// TwinCAT 3 PLC project aft_plc_harv_control
// ProgramVersion: 3.1.4026.12
// CompilerDefines: VISU_USEPROPERTYINFO
// libraries:
//   CmpBitmapPool, * (System)
//   Tc2_Standard, * (Beckhoff Automation GmbH)
//   Tc2_System, * (Beckhoff Automation GmbH)
//   Tc2_Utilities, * (Beckhoff Automation GmbH)
//   Tc3_Module, * (Beckhoff Automation GmbH)
//   VisuDialogs, * (System)
//   TcUnit,newest,www.tcunit.org
//   VisuSymbols,newest,System
// project tree:
//   DUTs/Device Level Structures/PD4/ PD4ControlWord.TcDUT, PD4OperationMode.TcDUT, PD4Polarity.TcDUT, PD4StatusWord.TcDUT, ST_PD4_HW.TcDUT, ST_PD4_IN.TcDUT, ST_PD4_OUT.TcDUT
//   DUTs/Device Level Structures/PD6/ PD6ControlWord.TcDUT, PD6OperationMode.TcDUT, PD6Polarity.TcDUT, PD6StatusWord.TcDUT, ST_PD6_IN.TcDUT, ST_PD6_HW.TcDUT, ST_PD6_OUT.TcDUT
//   DUTs/Device Level Structures/SevCon/ SevconControlWord.TcDUT, SevconStatusWord.TcDUT, ST_SEVCON_HW.TcDUT, ST_SEVCON_IN.TcDUT, ST_SEVCON_OUT.TcDUT
//   DUTs/ FrameSelect.TcDUT
//   DUTs/Message Structures/ ST_BINFILLER_MSG.TcDUT, ST_DRIVE_MSG.TcDUT, ST_ERROR_MSG.TcDUT
//   / GlobalTextList.TcGTLO, PlcTask.TcTTO, Visualization Manager.TcVMO (not stored), VISU_TASK.TcTTO
//   GVLs/ CONFIG.TcGVL, HARV.TcGVL, INDEX.TcGVL, IO.TcGVL, MOTORS.TcGVL, UI.TcGVL
//   POUs/Device Level Function Blocks/ FB_HYDRAULIC_VALVE.TcPOU, FB_PD4.TcPOU, FB_PD6.TcPOU, FB_SDO_READ.TcPOU, FB_SEVCON.TcPOU, FB_SDO_WRITE.TcPOU
//   POUs/ FB_READ_HW.TcPOU, FB_WRITE_HW.TcPOU, MAIN.TcPOU
//   POUs/Log Level Function Blocks/ FB_DRIVE_MSG_LOG.TcPOU, FB_ERROR_MSG_LOG.TcPOU, FB_TIMETRACKER.TcPOU
//   POUs/SubSystem Level Function Blocks/ FB_BINFILLER.TcPOU, FB_BIN_MANAGER.TcPOU, FB_CONVEYANCE.TcPOU, FB_DRIVE.TcPOU, FB_TILT.TcPOU
//   POUs/UI Level Function Blocks/ FB_FRAMESELECTOR.TcPOU
//   Test/ FB_DRIVE_TEST.TcPOU, FB_TILT_TEST.TcPOU, PRG_TEST.TcPOU
//   VISUs/ DriveSysTest.TcVIS, Icons.TcIPO (not stored), TiltControlTest.TcVIS
//   VISUs/Harv UI Components/Home Screen Components/ ChassisControls.TcVIS, DriveControls.TcVIS, LeftRobotStatus.TcVIS, RightRobotStatus.TcVIS, RobotStatusPopup.TcVIS
//   VISUs/Harv UI Components/Stats Screen Components/ LeftRobotStats.TcVIS, HarvStats.TcVIS, RightRobotStats.TcVIS
//   VISUs/Harv UI Components/Supervisor Screen Components/ BinFiller.TcVIS, ColorThreshold.TcVIS, Conveyance.TcVIS, LeftRobotControls.TcVIS, RightRobotControls.TcVIS
//   VISUs/Harv UI Components/ Home_Screen.TcVIS, Stats_Screen.TcVIS, StatusBar.TcVIS, Supervisor_Screen.TcVIS
// real-time tasks:
//   TASK PlcTask: cycle T#2ms, priority 20, ADS port 350
//   TASK VISU_TASK: cycle T#200000us, priority 30, ADS port 351
// I/O:
//   DEVICE Device 1 (EtherCAT), AmsNetId 5.123.135.181.2.1
//     Term 5 (EK1200) [EK1200-5000 EtherCAT Power supply (2A E-Bus)]
//       Term 9 (EL3064) [EL3064 4Ch. Ana. Input 0-10V] (disabled)
//       Term 6 (EL1018) [EL1018 8Ch. Dig. Input 24V, 10µs]
//       Term 7 (EL2008) [EL2008 8Ch. Dig. Output 24V, 0.5A]
//       Term 12 (EL6751) [EL6751 CANopen Master] (disabled)
//       Term 11 (EK1110) [EK1110 EtherCAT extension]
//     Left Steering (PD4-E601L42-E-65-1) [PD4-Ex-E-65-1 EtherCAT Drive (CoE)] (disabled)
//     Right Steering (PD4-E601L42-E-65-1) [PD4-Ex-E-65-1 EtherCAT Drive (CoE)] (disabled)
//   DEVICE Device 2 (EL6751) (disabled), AmsNetId 5.123.135.181.3.1
//     Drive Right (BorgWarner Gen4 (PMAC)Thu Feb  3 22:00:)
//     Drive Left (BorgWarner Gen4 (PMAC)Thu Feb  3 22:00:)
// variable links:
//   aft_plc_harv_control/aft_plc_harv_control Instance <-> Device 1 (EtherCAT)/Left Steering (PD4-E601L42-E-65-1)
//     PlcTask Inputs/MOTORS.SteerLeft.ActualPosition <-> Transmit PDO 1 Mapping Parameter/Position actual value
//     PlcTask Inputs/MOTORS.SteerLeft.OperationModeDisplay <-> Transmit PDO 1 Mapping Parameter/Modes of operation display
//     PlcTask Inputs/MOTORS.SteerLeft.StatusWord <-> Transmit PDO 1 Mapping Parameter/Statusword
//     PlcTask Outputs/MOTORS.SteerLeft.Accel <-> Receive PDO 2 Mapping Parameter/Accel
//     PlcTask Outputs/MOTORS.SteerLeft.ControlWord <-> Receive PDO 1 Mapping Parameter/Controlword
//     PlcTask Outputs/MOTORS.SteerLeft.Decel <-> Receive PDO 2 Mapping Parameter/Decel
//     PlcTask Outputs/MOTORS.SteerLeft.HomingMethod <-> Receive PDO 1 Mapping Parameter/Homing Method
//     PlcTask Outputs/MOTORS.SteerLeft.OperationMode <-> Receive PDO 1 Mapping Parameter/Modes of operation
//     PlcTask Outputs/MOTORS.SteerLeft.Polarity <-> Receive PDO 1 Mapping Parameter/Polarity
//     PlcTask Outputs/MOTORS.SteerLeft.ProfileVelocity <-> Receive PDO 2 Mapping Parameter/Profile velocity
//     PlcTask Outputs/MOTORS.SteerLeft.SubmodeSelect <-> Receive PDO 1 Mapping Parameter/Motor drive submode select
//     PlcTask Outputs/MOTORS.SteerLeft.TargetPosition <-> Receive PDO 2 Mapping Parameter/Target Position
//     PlcTask Outputs/MOTORS.SteerLeft.TargetVelocity <-> Receive PDO 3 Mapping Parameter/vl target velocity
//   aft_plc_harv_control/aft_plc_harv_control Instance <-> Device 1 (EtherCAT)/Right Steering (PD4-E601L42-E-65-1)
//     PlcTask Inputs/MOTORS.SteerRight.ActualPosition <-> Transmit PDO 1 Mapping Parameter/Position actual value
//     PlcTask Inputs/MOTORS.SteerRight.OperationModeDisplay <-> Transmit PDO 1 Mapping Parameter/Modes of operation display
//     PlcTask Inputs/MOTORS.SteerRight.StatusWord <-> Transmit PDO 1 Mapping Parameter/Statusword
//     PlcTask Outputs/MOTORS.SteerRight.Accel <-> Receive PDO 2 Mapping Parameter/Accel
//     PlcTask Outputs/MOTORS.SteerRight.ControlWord <-> Receive PDO 1 Mapping Parameter/Controlword
//     PlcTask Outputs/MOTORS.SteerRight.Decel <-> Receive PDO 2 Mapping Parameter/Decel
//     PlcTask Outputs/MOTORS.SteerRight.HomingMethod <-> Receive PDO 1 Mapping Parameter/Homing Method
//     PlcTask Outputs/MOTORS.SteerRight.OperationMode <-> Receive PDO 1 Mapping Parameter/Modes of operation
//     PlcTask Outputs/MOTORS.SteerRight.Polarity <-> Receive PDO 1 Mapping Parameter/Polarity
//     PlcTask Outputs/MOTORS.SteerRight.ProfileVelocity <-> Receive PDO 2 Mapping Parameter/Profile velocity
//     PlcTask Outputs/MOTORS.SteerRight.SubmodeSelect <-> Receive PDO 1 Mapping Parameter/Motor drive submode select
//     PlcTask Outputs/MOTORS.SteerRight.TargetPosition <-> Receive PDO 2 Mapping Parameter/Target Position
//     PlcTask Outputs/MOTORS.SteerRight.TargetVelocity <-> Receive PDO 3 Mapping Parameter/vl target velocity
//   aft_plc_harv_control/aft_plc_harv_control Instance <-> Device 1 (EtherCAT)/Term 5 (EK1200)/Term 6 (EL1018)
//     PlcTask Inputs/IO.DI_SLICE_0[{0..7}] <-> Channel {1..8}/Input  (8 links)
//   aft_plc_harv_control/aft_plc_harv_control Instance <-> Device 1 (EtherCAT)/Term 5 (EK1200)/Term 7 (EL2008)
//     PlcTask Outputs/IO.DO_SLICE_0[{0..7}] <-> Channel {1..8}/Output  (8 links)
//   aft_plc_harv_control/aft_plc_harv_control Instance <-> Device 1 (EtherCAT)/Term 5 (EK1200)/Term 9 (EL3064)
//     PlcTask Inputs/IO.AI_SLICE_0[{0..3}] <-> AI Standard Channel {1..4}/Value  (4 links)
//   aft_plc_harv_control/aft_plc_harv_control Instance <-> Device 2 (EL6751)/Drive Left (BorgWarner Gen4 (PMAC)Thu Feb  3 22:00:)
//     PlcTask Inputs/MOTORS.DriveLeft.ActualVelocity <-> TxPDO 1/Inputs/Actual Velocity
//     PlcTask Inputs/MOTORS.DriveLeft.AnalogIn{1..4} <-> TxPDO 3/Inputs/Analog In {1..4}  (4 links)
//     PlcTask Inputs/MOTORS.DriveLeft.BatteryCurrent <-> TxPDO 2/Inputs/Battery Current
//     PlcTask Inputs/MOTORS.DriveLeft.BatteryVoltage <-> TxPDO 2/Inputs/Battery Voltage
//     PlcTask Inputs/MOTORS.DriveLeft.CapacitorVoltage <-> TxPDO 2/Inputs/Capacitor Voltage
//     PlcTask Inputs/MOTORS.DriveLeft.HeatsinkTemp <-> TxPDO 2/Inputs/Heatsink Temp
//     PlcTask Inputs/MOTORS.DriveLeft.StatusWord <-> TxPDO 1/Inputs/Status Word
//     PlcTask Outputs/MOTORS.DriveLeft.BrakeOutput <-> RxPDO 3/Outputs/Brake
//     PlcTask Outputs/MOTORS.DriveLeft.ContactorOutput <-> RxPDO 3/Outputs/Power Contactor
//     PlcTask Outputs/MOTORS.DriveLeft.ControlWord <-> RxPDO 1/Outputs/Control Word
//     PlcTask Outputs/MOTORS.DriveLeft.TargetVelocity <-> RxPDO 1/Outputs/Target Velocity

CONFIGURATION aft_plc_harv_control
    RESOURCE PLC ON TwinCAT3
        TASK PlcTask(INTERVAL := T#2ms, PRIORITY := 20);
        TASK VISU_TASK(INTERVAL := T#200000us, PRIORITY := 30);
        PROGRAM MAIN WITH PlcTask : MAIN;
        PROGRAM PRG_TEST WITH PlcTask : PRG_TEST;
        PROGRAM VisuElems_Visu_Prg WITH VISU_TASK : VisuElems.Visu_Prg;
    END_RESOURCE
END_CONFIGURATION

// ---- DUTs/Device Level Structures/PD4/PD4ControlWord.TcDUT
{attribute 'qualified_only'}
{attribute 'strict'}
TYPE PD4ControlWord :
(
	Shutdown := 6,					// 2#0000_0110	
	SwitchOn := 7,					// 0xxx 0111 (Trasition from Ready to Switch On -> Switched On)
	SwitchOnOperationEnable := 15,	// 0xxx 1111 (Switch On and Enable Operation)
	StartHoming:= 16,
	PulseInhibit := 0,				// 0xxx xx0x (activate quick stop and disable)
	QuickStop := 2,					// 0xxx x01x
	DisableOperation := 7,			// 0xxx 0111 (Transition from OpEnable -> Switched On)
	EnableOperation := 2#00101111,			// 0x1x 1111
	FaultReset := 128,				// 1xxx xxxx
	StartMove := 2#00010000,				// xxx1 1111
	AbsoluteMotion := 2#00100000
	// Positive := 64,					// x1xx xxxx
	// Negative :=	0					// x0xx xxxx
)BYTE;
END_TYPE

// ---- DUTs/Device Level Structures/PD4/PD4OperationMode.TcDUT
{attribute 'qualified_only'}
{attribute 'strict'}
TYPE PD4OperationMode :
(
	ProfilePositionMode := 1,
	VelocityMode := 2,
	ProfileVelocityMode := 3,
	ProfileTorqueMode := 4,
	HomingMode := 6,
	CyclicSyncPositionMode := 8
)SINT;
END_TYPE

// ---- DUTs/Device Level Structures/PD4/PD4Polarity.TcDUT
{attribute 'qualified_only'}
{attribute 'strict'}
TYPE PD4Polarity :
(
	Positive := 64,
	Negative := 0
)USINT;
END_TYPE

// ---- DUTs/Device Level Structures/PD4/PD4StatusWord.TcDUT
{attribute 'qualified_only'}
{attribute 'strict'}
TYPE PD4StatusWord :
(
	NotReadyToSwitchOn := 0,	// x0xx 0000
	SwitchOnDisabled := 64,		// x1xx 0000
	ReadyToSwitchOn := 33,		// 1000 0010 0011 0001 (0x8231)
	SwitchedOn := 35,			// 1000 0010 0011 0011 (0x8233)
	OperationEnabled := 39,		// x01x 0111
	QuickStopActive := 7,		// x00x 0111
	Fault := 8,					// x0xx 1000
	TargetReached := 1024,		// 0000 0100 0000 0000 (bit 10)
	HomingComplete := 5120,		// 0001 0100 0000 0000 (bit 10 and 12)
	TargetPositionAccepted := 4096		
)UINT;
END_TYPE

// ---- DUTs/Device Level Structures/PD4/ST_PD4_HW.TcDUT
TYPE ST_PD4_HW :
STRUCT
	StatusWord 				AT %I* : UINT; 
	OperationModeDisplay 	AT %I* : SINT;
	ActualPosition 			AT %I* : DINT;
	ActualVelocity 			AT %I* : INT;
	
	
	ControlWord 	AT %Q* : UINT;
	HomingMethod 	AT %Q* : USINT;
	TargetVelocity 	AT %Q* : INT;
	ProfileVelocity AT %Q* : UDINT;
	Accel 			AT %Q* : UDINT;				
	Decel 			AT %Q* : UDINT;				
	SubmodeSelect	AT %Q* : UDINT;	
	OperationMode 	AT %Q* : SINT;	
	TargetPosition 	AT %Q* : DINT;		
	Polarity 		AT %Q* : USINT;		
END_STRUCT
END_TYPE

// ---- DUTs/Device Level Structures/PD4/ST_PD4_IN.TcDUT
TYPE ST_PD4_IN :
STRUCT
	StatusWord 				: UINT;
	ActualPosition 			: DINT;
	ActualVelocity 			: REAL;
	OperationModeDisplay 	: SINT;
END_STRUCT
END_TYPE

// ---- DUTs/Device Level Structures/PD4/ST_PD4_OUT.TcDUT
TYPE ST_PD4_OUT :
STRUCT
	ControlWord 	: UINT;
	HomingMethod 	: USINT;
	TargetVelocity 	: INT;		// target velocity while in profile velocity mode
	ProfileVelocity : UDINT;	// target velocity while in profile position mode
	Accel 			: UDINT;
	Decel 			: UDINT;
	TargetPosition	: DINT;
	SubmodeSelect 	: UDINT;
	OperationMode 	: SINT;
	Polarity		: USINT;
END_STRUCT
END_TYPE

// ---- DUTs/Device Level Structures/PD6/PD6ControlWord.TcDUT
{attribute 'qualified_only'}
{attribute 'strict'}
TYPE PD6ControlWord :
(
	Shutdown := 6,					// 2#0000_0110	
	SwitchOn := 7,					// 0xxx 0111 (Trasition from Ready to Switch On -> Switched On)
	SwitchOnOperationEnable := 15,	// 0xxx 1111 (Switch On and Enable Operation)
	StartHoming:= 16,
	PulseInhibit := 0,				// 0xxx xx0x (activate quick stop and disable)
	QuickStop := 2,					// 0xxx x01x
	DisableOperation := 7,			// 0xxx 0111 (Transition from OpEnable -> Switched On)
	EnableOperation := 15,			// 0xxx 1111
	FaultReset := 128,				// 1xxx xxxx
	StartMove := 2#00010000,				// xxx1 1111
	AbsoluteMotion := 2#00100000			// xxx1 1111
	// Positive := 64,					// x1xx xxxx
	// Negative :=	0					// x0xx xxxx
)BYTE;
END_TYPE

// ---- DUTs/Device Level Structures/PD6/PD6OperationMode.TcDUT
{attribute 'qualified_only'}
{attribute 'strict'}
TYPE PD6OperationMode :
(
	ProfilePositionMode := 1,
	VelocityMode := 2,
	ProfileVelocityMode := 3,
	ProfileTorqueMode := 4,
	HomingMode := 6,
	CyclicSyncPositionMode := 8
)SINT;
END_TYPE

// ---- DUTs/Device Level Structures/PD6/PD6Polarity.TcDUT
{attribute 'qualified_only'}
{attribute 'strict'}
TYPE PD6Polarity :
(
	Positive := 64,
	Negative := 0
)USINT;
END_TYPE

// ---- DUTs/Device Level Structures/PD6/PD6StatusWord.TcDUT
{attribute 'qualified_only'}
{attribute 'strict'}
TYPE PD6StatusWord :
(
	NotReadyToSwitchOn := 0,	// x0xx 0000
	SwitchOnDisabled := 64,		// x1xx 0000
	ReadyToSwitchOn := 33,		// 1000 0010 0011 0001 (0x8231)
	SwitchedOn := 35,			// 1000 0010 0011 0011 (0x8233)
	OperationEnabled := 39,		// x01x 0111
	QuickStopActive := 7,		// x00x 0111
	Fault := 8,					// x0xx 1000
	TargetReached := 1024,		// 0000 0100 0000 0000 (bit 10)
	HomingComplete := 5120,		// 0001 0100 0000 0000 (bit 10 and 12)
	TargetPositionAccepted := 4096		
)UINT;
END_TYPE

// ---- DUTs/Device Level Structures/PD6/ST_PD6_IN.TcDUT
TYPE ST_PD6_IN :
STRUCT
	StatusWord 				: UINT; 
	OperationModeDisplay 	: SINT;
	ActualPosition 			: DINT;
	ActualVelocity 			: INT;
	ActiveCurrent			: REAL;
END_STRUCT
END_TYPE

// ---- DUTs/Device Level Structures/PD6/ST_PD6_HW.TcDUT
TYPE ST_PD6_HW :
STRUCT
	StatusWord 				AT %I* : UINT; 
	OperationModeDisplay 	AT %I* : SINT;
	ActualPosition 			AT %I* : DINT;
	ActualVelocity 			AT %I* : INT;
	
	
	ControlWord 	AT %Q* : UINT;
	HomingMethod 	AT %Q* : USINT;
	TargetVelocity 	AT %Q* : INT;
	ProfileVelocity AT %Q* : UDINT;
	Accel 			AT %Q* : UDINT;				
	Decel 			AT %Q* : UDINT;				
	SubmodeSelect	AT %Q* : UDINT;	
	OperationMode 	AT %Q* : SINT;	
	TargetPosition 	AT %Q* : DINT;		
	Polarity 		AT %Q* : USINT;		
END_STRUCT
END_TYPE

// ---- DUTs/Device Level Structures/PD6/ST_PD6_OUT.TcDUT
TYPE ST_PD6_OUT :
STRUCT
	ControlWord 	: UINT;
	HomingMethod 	: USINT;
	TargetVelocity 	: INT;
	ProfileVelocity : UDINT;
	Accel 			: UDINT;				
	Decel 			: UDINT;				
	SubmodeSelect	: UDINT;	
	OperationMode 	: SINT;	
	TargetPosition 	: DINT;		
	Polarity 		: USINT;	
END_STRUCT
END_TYPE

// ---- DUTs/Device Level Structures/SevCon/SevconControlWord.TcDUT
{attribute 'qualified_only'}
{attribute 'strict'}
TYPE SevconControlWord :
(
	Shutdown			:= 2#00000110,
	SwitchOn			:= 2#00000111,
	DisableVoltage		:= 2#00000000,
	QuickStop			:= 2#00000010,
	DisableOperation	:= 2#00000111,
	EnableOperation		:= 2#00001111,
	FaultReset			:= 2#00010000
)BYTE;
END_TYPE

// ---- DUTs/Device Level Structures/SevCon/SevconStatusWord.TcDUT
{attribute 'qualified_only'}
{attribute 'strict'}
TYPE SevconStatusWord :
(
	SwitchOnDisabled	:= 2#01000000,
	ReadyToSwitchon		:= 2#00100001,
	Switchedon			:= 2#00100011,
	OperationEnabled	:= 2#00100111,
	QuickStopActive		:= 2#00000111,
	FaultReactionActive	:= 2#00001111,
	Fault				:= 2#00001000
)BYTE;
END_TYPE

// ---- DUTs/Device Level Structures/SevCon/ST_SEVCON_HW.TcDUT
TYPE ST_SEVCON_HW :
STRUCT
	(*Inputs to PLC from Sevcon*)
	StatusWord 				AT %I* : UINT;
	OperationModeDisplay 	AT %I* : SINT;
	ActualVelocity 			AT %I* : UDINT;
	BatteryVoltage			AT %I* : UINT;
	BatteryCurrent			AT %I* : UINT;
	CapacitorVoltage		AT %I* : UINT;
	HeatsinkTemp			AT %I* : USINT;
	AnalogIn1				AT %I* : UINT;
	AnalogIn2				AT %I* : UINT;
	AnalogIn3				AT %I* : UINT;
	AnalogIn4				AT %I* : UINT;
	
	
	(*Outputs to Sevcon from PLC*)
	ControlWord 	AT %Q* : UINT;
	OperationMode 	AT %Q* : SINT;
	TargetVelocity	AT %Q* : UDINT;
	Accel			AT %Q* : UINT;
	Decel			AT %Q* : UINT;
	BrakeOutput		AT %Q* : UINT;
	ContactorOutput	AT %Q* : UINT;
END_STRUCT
END_TYPE

// ---- DUTs/Device Level Structures/SevCon/ST_SEVCON_IN.TcDUT
TYPE ST_SEVCON_IN :
STRUCT
	StatusWord 				: UINT;
	OperationModeDisplay 	: SINT;
	ActualVelocity 			: UDINT;
	BatteryVoltage			: UINT;
	BatteryCurrent			: UINT;
	CapacitorVoltage		: UINT;
	HeatsinkTemp			: UINT;
	AnalogIn1				: UINT;
	AnalogIn2				: UINT;
	AnalogIn3				: UINT;
	AnalogIn4				: UINT;
END_STRUCT
END_TYPE

// ---- DUTs/Device Level Structures/SevCon/ST_SEVCON_OUT.TcDUT
TYPE ST_SEVCON_OUT :
STRUCT
	ControlWord 	: UINT;
	OperationMode 	: SINT;
	TargetVelocity	: UDINT;
	Accel			: UINT;
	Decel			: UINT;
	BrakeOutput		: UINT;
	ContactorOutput	: UINT;
	PreCharge		: UINT;
END_STRUCT
END_TYPE

// ---- DUTs/FrameSelect.TcDUT
{attribute 'qualified_only'}
{attribute 'strict'}
TYPE FrameSelect :
(
	Status	:= 1,
	Warning := 2,
	Error	:= 3
)INT;
END_TYPE

// ---- DUTs/Message Structures/ST_BINFILLER_MSG.TcDUT
{attribute 'pack_mode' := '1'}
TYPE ST_BINFILLER_MSG :
STRUCT
END_STRUCT
END_TYPE

// ---- DUTs/Message Structures/ST_DRIVE_MSG.TcDUT
{attribute 'pack_mode' := '1'}
TYPE ST_DRIVE_MSG :
STRUCT
	TimeStamp			: DT;
	LeftVelocity		: INT;
	RightVelocity		: INT;
	LeftSteeringAngle	: LREAL;
	RightSteeringAngle	: LREAL;
	LeftCurrent			: REAL;
	RightCurrent		: REAL;
	LeftStatusCode		: UINT;
	RightStatusCode		: UINT;
END_STRUCT
END_TYPE

// ---- DUTs/Message Structures/ST_ERROR_MSG.TcDUT
{attribute 'pack_mode' := '1'}
TYPE ST_ERROR_MSG :
STRUCT
	Timestamp	: DT;
	Location	: STRING;
	ErrorCode	: INT;
	Description	: STRING;
END_STRUCT
END_TYPE

// ---- GVLs/CONFIG.TcGVL
{attribute 'qualified_only'}
VAR_GLOBAL
	
	DriveWheelWidth			: REAL := 8.0;
	
	SteeringWheelWidth		: REAL := 5.0;
	WheelBase				: REAL := 137.0;		// Distance between the drive wheels and steering wheels center to center
	FrontTrackWidth			: REAL := 60;		// Distance between the two drive wheels center to center
	RearTrackWidth			: REAL := 72;		// inches
	CasterOffset			: REAL := 8.0;		// Distance between wheel center and rotation center on the steering axes
	
	SevCon_Port				: ARRAY[0..1] OF WORD := [16#1001, 16#1002];	// Drive Right, Drive Left
END_VAR

// ---- GVLs/HARV.TcGVL
{attribute 'qualified_only'}
VAR_GLOBAL
	(*Log Level Function Blocks*)
	ErrorLog	: FB_ERROR_MSG_LOG;
	DriveLog	: FB_DRIVE_MSG_LOG;
	TimeTracker	: FB_TIMETRACKER;
	
	(*SubSystem Level Function Blocks*)
	DriveSys	: FB_DRIVE;
	TiltControl	: FB_TILT;
	BinFiller	: FB_BINFILLER;
	BinManager	: FB_BIN_MANAGER;
	Conveyance	: FB_CONVEYANCE;
	
	(*Device Level Function Blocks*)
	ReadHw		: FB_READ_HW;
	WriteHw		: FB_WRITE_HW;
	
	(*System Level Function Blocks*)
	SystemReboot	: NT_REBOOT;
END_VAR

// ---- GVLs/INDEX.TcGVL
{attribute 'qualified_only'}
VAR_GLOBAL
	(*SEVCON Indexes that will likely be used by the SDO Read/Write function blocks*)
	SpeedControlGains	: DWORD := 16#4651;
	PasswordEntry		: DWORD := 16#5000;
	PasswordKey			: DWORD := 16#5001;	
	NmtState			: DWORD := 16#5110;
	PreChargeActivate	: DWORD := 16#5180;
	FinalPreChargeLevel	: DWORD := 16#5820;
	MinPreChargeLevel	: DWORD := 16#5821;
END_VAR

// ---- GVLs/IO.TcGVL
{attribute 'qualified_only'}
VAR_GLOBAL
	AI_SLICE_0 AT %I* : ARRAY[0..3] OF INT;
	DI_SLICE_0 AT %I* : ARRAY[0..7] OF BOOL;
	
	DO_SLICE_0 AT %Q* : ARRAY[0..7] OF BOOL;
END_VAR

// ---- GVLs/MOTORS.TcGVL
{attribute 'qualified_only'}
VAR_GLOBAL
	DriveLeft	: ST_SEVCON_HW;
	DriveRight	: ST_SEVCON_HW;
//	DriveLeft	: ST_PD6_HW;
//	DriveRight	: ST_PD6_HW;
//	SteerLeft_PD6	: ST_PD6_HW;
//	SteerRight_PD6	: ST_PD6_HW;
	SteerLeft	: ST_PD4_HW;
	SteerRight	: ST_PD4_HW;
END_VAR

// ---- GVLs/UI.TcGVL
{attribute 'qualified_only'}
VAR_GLOBAL
	FrameSelector	: FB_FRAMESELECTOR;
	PickButton		: BOOL;
	EStop			: BOOL;
END_VAR

// ---- POUs/MAIN.TcPOU
PROGRAM MAIN
VAR
	Error			: BOOL;
	SystemReboot	: NT_REBOOT;
	Reboot			: BOOL;
	MsgUpdateTimer	: TON;
	MsgUpdatePeriod	: TIME := T#50MS;
	TimerResetDelay	: INT := 25;
	TimerResetCounter	: INT;
	Version			: REAL := 1.0;
	
	State			: (DEFAULT, INIT, IDLE, RUN, ERROR);
	PrevState		: (DEFAULT, INIT, IDLE, RUN, ERROR);
	StateEntry 		: BOOL;
END_VAR

Harv.ReadHw();

MsgUpdateTimer.PT := MsgUpdatePeriod;

IF PrevState <> State THEN
	StateEntry := TRUE;
	PrevState := State;
ELSE
	StateEntry := FALSE;
END_IF

CASE State OF
	DEFAULT:
		//
	INIT:
		//
	IDLE:
		//
	RUN:
		//
	ERROR:
		//
END_CASE

//IF Error THEN
//	HARV.ErrorLog.AddMsg(TimeStamp := Harv.TimeTracker.TimeStamp, Location := 'MAIN', ErrorCode := 1234, Description := 'TEST');
//	Error := FALSE;
//END_IF

IF MsgUpdateTimer.Q THEN
	TimerResetCounter := TimerResetCounter + 1;
	IF TimerResetCounter = TimerResetDelay THEN
		TimerResetCounter := 0;
		MsgUpdateTimer.IN := FALSE;
	END_IF
ELSE
	TimerResetCounter := 0;
	MsgUpdateTimer.IN := TRUE;
END_IF

SystemReboot(NETID := '', START := Reboot);

MsgUpdateTimer();
Harv.TimeTracker();
Harv.DriveSys();
Harv.TiltControl();
Harv.WriteHw();

END_PROGRAM

// ---- Test/PRG_TEST.TcPOU
PROGRAM PRG_TEST
VAR
	Drive_Test	: FB_DRIVE_TEST;
END_VAR

TcUnit.RUN();

END_PROGRAM

// ---- Test/FB_DRIVE_TEST.TcPOU
FUNCTION_BLOCK FB_DRIVE_TEST EXTENDS TcUnit.FB_TestSuite
VAR_INPUT
END_VAR
VAR_OUTPUT
END_VAR
VAR
END_VAR

SteerAngleTest();
DiffDriveTest();

METHOD DiffDriveTest : REFERENCE TO FB_Test
VAR
	
END_VAR
TEST('DifferentialDriveTest');



TEST_FINISHED();
END_METHOD

METHOD SteerAngleTest : REFERENCE TO FB_Test
VAR
	Drive	: FB_DRIVE;
	AngleInput			: LREAL := 45;
	LeftAngleCalc		: LREAL;
	RightAngleCalc		: LREAL;	
	LeftAngleExpected	: LREAL := 38.89;
	RightAngleExpected	: LREAL := 51.03;
END_VAR
TEST('SteerAngleTest');

(*Zero Steering Angle*)
Drive.CalcWheelAngle(0);
LeftAngleCalc := Drive.SteerLeftAngleTest;
RightAngleCalc := Drive.SteerRightAngleTest;
			
AssertEquals_LREAL(Expected := 0,
				Actual := LeftAngleCalc,
				Delta := 0.1,
				Message := 'Left Angle 0 Calculation Incorrect');
				
AssertEquals_LREAL(Expected := 0,
				Actual := RightAngleCalc,
				Delta := 0.1,
				Message := 'Right Angle 0 Calculation Incorrect');

(*45 Degree Steering Angle*)				
Drive.CalcWheelAngle(AngleInput);
LeftAngleCalc := Drive.SteerLeftAngleTest;
RightAngleCalc := Drive.SteerRightAngleTest;

AssertEquals_LREAL(Expected := LeftAngleExpected,
				Actual := LeftAngleCalc,
				Delta := 0.1,
				Message := 'Left Angle 45 Calculation Incorrect');
				
AssertEquals_LREAL(Expected := RightAngleExpected,
				Actual := RightAngleCalc,
				Delta := 0.1,
				Message := 'Right Angle 45 Calculation Incorrect');

(*-45 Degree Steering Angle*)			
Drive.CalcWheelAngle(-AngleInput);
LeftAngleCalc := Drive.SteerLeftAngleTest;
RightAngleCalc := Drive.SteerRightAngleTest;

AssertEquals_LREAL(Expected := -RightAngleExpected,
				Actual := LeftAngleCalc,
				Delta := 0.1,
				Message := 'Left Angle -45 Calculation Incorrect');
				
AssertEquals_LREAL(Expected := -LeftAngleExpected,
				Actual := RightAngleCalc,
				Delta := 0.1,
				Message := 'Right Angle -45 Calculation Incorrect');
				
(*Positive Max Steering Angle*)

(*Negative Max Steering Angle*)

(*Positive Out of Range Steering Angle*)

(*Negative Out of Range Steering Angle*)
			
TEST_FINISHED();
END_METHOD

END_FUNCTION_BLOCK

// ---- POUs/SubSystem Level Function Blocks/FB_DRIVE.TcPOU
FUNCTION_BLOCK FB_DRIVE
VAR_INPUT
	DriveLeftIN			: ST_SEVCON_IN;
	DriveRightIN		: ST_SEVCON_IN;
//	SteerLeftIN			: ST_PD6_IN;
//	SteerRightIN		: ST_PD6_IN;
	SteerLeftIN			: ST_PD4_IN;
	SteerRightIN		: ST_PD4_IN;
	
	JoyStick_X			: INT;
	JoyStick_Y			: INT;
	JoyStick_Button		: INT;
	ManualDriveEnable	: BOOL;			// Dead man switch on joystick controls
	AutoDriveEnable		: BOOL;			// Likely controlled by python
	ErrorReset			: BOOL;
	
	AutoDriveSpeedCommand	: DINT := 50;
	JohnButtonInput		: BOOL;
END_VAR
VAR_OUTPUT
	DriveLeft	: FB_SEVCON;
	DriveRight	: FB_SEVCON;
//	SteerLeft	: FB_PD6;
//	SteerRight	: FB_PD6;
	SteerLeft	: FB_PD4;
	SteerRight	: FB_PD4;
	
	(*Outputs for unit testing*)
	SteerLeftAngleTest	: LREAL;
	SteerRightAngleTest	: LREAL;

	Error		: BOOL;
	ErrorCode	: INT;
	Ready		: BOOL;
END_VAR
VAR
	State		: (DEFAULT, INIT, IDLE, MANUAL, AUTO, ERROR);
	PrevState	: (DEFAULT, INIT, IDLE, MANUAL, AUTO, ERROR);
	StateEntry 	: BOOL;
	TimeInState	: TIME;
	
	LeftVelCommand	: LREAL;
	LeftVelActual	: LREAL;
	LeftPosActual	: DINT;
	RightVelCommand	: LREAL;
	RightVelActual	: LREAL;
	RightPosActual	: DINT;
	DriveVelInput	: LREAL;
				// Check variable type here, will be in acres / hour
	AutoDriveSpeedActual	: DINT := 45;			// in Acres/hour
	
	SteeringAngleInput		: LREAL;		// unit should be degrees, max range is +/- 89 degrees
	ICC_R					: LREAL;		// instantaneous radius of curvature calculated from steering angle
	LeftWheelAngleCommand	: LREAL;
	LeftWheelAngleActual	: LREAL;
	RightWheelAngleCommand	: LREAL;
	RightWheelAngleActual	: LREAL;
	
	DriveMsgUpdateTimer		: TON;
	DriveMsgUpdatePeriod	: TIME := T#5S;
END_VAR
VAR CONSTANT
	MaxDriveSpeed			: REAL := 1000;		// mm/s
	MaxSteeringAngle		: REAL := 75.0;		// degrees
	JoyStickMaxVal			: INT := 16300;	// raw analog value at extreme
	JoyStickCenter			: INT := 8150;
	DeadBand_X				: INT := 150;		// ~10% or +/- 1V
	DeadBand_Y				: INT := 150;		// ~10% or +/- 1V
	DriveWheelDiameter		: REAL := 762;		// in mm = 30 inches
	DriveWheelEncoderRes	: DINT := 1000;		// was 4000
	DriveWheelGearRatio		: INT := 1;
	SteeringWheelDiameter	: REAL := 660.4;	// in mm = 26 inches
	SteeringEncoderRes		: DINT := 4000;
	SteeringGearRatio		: INT := 14;
	SteeringVel				: UDINT := 500;
	SteeringAcc				: UDINT := 1000;
	SteeringDec				: UDINT := 1000;
	DriveAcc				: UDINT := 1000;
	DriveDec				: UDINT := 10000;
END_VAR

(*DRIVE SYSTEM CONTROL FUNCTION BLOCK
INPUTS:
	- Joystick values in X and Y direction in Manual Drive Mode
	- Deadman switch input for manual mode activation and safety
	- Drive Velocity and Steering Angle from Python in Auto Drive Mode
	- Device status from Sevcons, PD6s and other motion devices

OUTPUTS:
	- Target Velocity commands to SEVCONs for drive speed control
	- Target Position commands to PD6/4s for steering angle control
	- Device status info and function block state*)

IF State <> PrevState THEN
	StateEntry := TRUE;
	PrevState := State;
ELSE
	StateEntry := FALSE;
END_IF

CASE State OF
	DEFAULT:
		IF StateEntry THEN
			TimeInState := T#0MS;
		END_IF
		
		State := INIT;
		
	INIT:
		IF StateEntry THEN
			DriveMsgUpdateTimer.PT := DriveMsgUpdatePeriod;
			TimeInState := T#0MS;
		END_IF
		
		SteerLeft.SetMotionProfile(SteeringVel, SteeringAcc, SteeringDec);
		SteerRight.SetMotionProfile(SteeringVel, SteeringAcc, SteeringDec);
		
		DriveRight.Self := 1;
		DriveLeft.Self := 2;
		
		IF (DriveLeft.Ready) THEN
			Ready := TRUE;
			State := IDLE;
		END_IF
		
//		IF (SteerLeft.Ready AND SteerRight.Ready AND DriveLeft.Ready AND DriveRight.Ready) THEN
//			Ready := TRUE;
//			State := IDLE;
//		END_IF
		
	IDLE:
		IF StateEntry THEN
			TimeInState := T#0MS;
		END_IF
		
		ReadButton();
		
		IF ManualDriveEnable AND Ready THEN
			State := MANUAL;
		ELSIF AutoDriveEnable AND Ready THEN
			State := AUTO;
		END_IF

	MANUAL:
		IF StateEntry THEN
			TimeInState := T#0MS;
			DriveLeft.Enable := TRUE;
			// DriveRight.Enable := TRUE;
			SteerLeft.Enable := TRUE;
			SteerRight.Enable := TRUE;
		END_IF
		
		(*Reads joystick in X direction, scales for steering angle and implements deadband limits*)
		IF (JoyStick_X > (JoyStickCenter + DeadBand_X)) THEN
			SteeringAngleInput := (INT_TO_REAL(JoyStick_X - (JoyStickCenter + DeadBand_X)) / (JoyStickCenter - DeadBand_X)) * MaxSteeringAngle;
		ELSIF (JoyStick_X < (JoyStickCenter - DeadBand_X)) THEN
			SteeringAngleInput := (INT_TO_REAL(JoyStick_X -(JoyStickCenter - DeadBand_X)) / (JoyStickCenter - DeadBand_X)) * MaxSteeringAngle;
		ELSE
			SteeringAngleInput := 0;
		END_IF
		
		(*Reads joystick in Y direction, scales for drive speed and implements deadband limits*)
		IF (JoyStick_Y > (JoyStickCenter + DeadBand_Y)) THEN
			DriveVelInput := (INT_TO_REAL(JoyStick_Y - (JoyStickCenter + DeadBand_Y)) / (JoyStickCenter - DeadBand_Y)) * MaxDriveSpeed;
		ELSIF (JoyStick_Y < (JoyStickCenter - DeadBand_Y)) THEN
			DriveVelInput := (INT_TO_REAL(JoyStick_Y - (JoyStickCenter - DeadBand_Y)) / (JoyStickCenter - DeadBand_Y)) * MaxDriveSpeed;
		ELSE
			DriveVelInput := 0;
		END_IF
		
		(*Calculates wheel angles needed to achieve the commanded steering angle*)
		CalcWheelAngle(SteeringAngleInput);					
		
		(*Calculates differential velocities of the left and right wheels*)
		CalcDiffVelocity(DriveVelInput);				
		
		(*Sets the Sevcon target velocities equal to the calculated values and applies unit scaling*)
		DriveLeft.TargetVelocity := LREAL_TO_UDINT((LeftVelCommand / (3.14 * DriveWheelDiameter)) * DriveWheelGearRatio * DriveWheelEncoderRes);
		DriveRight.TargetVelocity := LREAL_TO_UDINT((RightVelCommand / (3.14 * DriveWheelDiameter)) * DriveWheelGearRatio * DriveWheelEncoderRes);
		
		(*Sets the PD4 steering motors to the correct positions*)
		SteerLeft.TargetPosition := -LREAL_TO_DINT(LeftWheelAngleCommand * ((SteeringEncoderRes * SteeringGearRatio) / 360));		// Negative for motor dir
		SteerRight.TargetPosition := -LREAL_TO_DINT(RightWheelAngleCommand * ((SteeringEncoderRes * SteeringGearRatio) / 360));		// Negative for motor dir
		
		ReadButton();
		
		IF NOT ManualDriveEnable THEN
			DriveLeft.TargetVelocity := 0;
			DriveRight.TargetVelocity := 0;
			DriveLeft.Enable := FALSE;
			DriveRight.Enable := FALSE;
			SteerLeft.Enable := FALSE;
			SteerRight.Enable := FALSE;
			State := IDLE;
		END_IF
		
	AUTO:
		IF StateEntry THEN
			TimeInState := T#0MS;
			DriveLeft.Enable := TRUE;
			DriveRight.Enable := TRUE;
			SteerLeft.Enable := TRUE;
			SteerRight.Enable := TRUE;
		END_IF
		
		(*Calculates wheel angles needed to achieve the commanded steering angle*)
		CalcWheelAngle(SteeringAngleInput);					
		
		(*Calculates differential velocities of the left and right wheels*)
		CalcDiffVelocity(DriveVelInput);	
		
		(*Sets the Sevcon target velocities equal to the calculated values and applies unit scaling*)
		DriveLeft.TargetVelocity := LREAL_TO_UDINT((LeftVelCommand / (3.14 * DriveWheelDiameter)) * DriveWheelGearRatio * DriveWheelEncoderRes);
		DriveRight.TargetVelocity := LREAL_TO_UDINT((RightVelCommand / (3.14 * DriveWheelDiameter)) * DriveWheelGearRatio * DriveWheelEncoderRes);
		
		(*Sets the PD6 steering motors to the correct positions*)
		SteerLeft.TargetPosition := LREAL_TO_DINT(LeftWheelAngleCommand * ((SteeringEncoderRes * SteeringGearRatio) / 360));
		SteerRight.TargetPosition := LREAL_TO_DINT(RightWheelAngleCommand * ((SteeringEncoderRes * SteeringGearRatio) / 360));
		
		IF NOT AutoDriveEnable THEN
			DriveLeft.TargetVelocity := 0;
			DriveRight.TargetVelocity := 0;
			DriveLeft.Enable := FALSE;
			DriveRight.Enable := FALSE;
			SteerLeft.Enable := FALSE;
			SteerRight.Enable := FALSE;
			State := IDLE;
		END_IF
		
	ERROR:
		IF StateEntry THEN
			Error := TRUE;
			Ready := FALSE;
			HARV.ErrorLog.AddMsg(TimeStamp := HARV.TimeTracker.TimeStamp, Location := 'DRIVE', ErrorCode := 9999, Description := 'Drive Test');
			TimeInState := T#0MS;
		END_IF
		
		IF ErrorReset THEN
			DriveLeft.ErrorReset := TRUE;
			DriveRight.ErrorReset := TRUE;
			SteerLeft.ErrorReset := TRUE;
			SteerRight.ErrorReset := TRUE;
			IF (NOT DriveLeft.Error) AND (NOT DriveRight.Error) AND (NOT SteerLeft.Error) AND (NOT SteerRight.Error) THEN
				Error := FALSE;
				ErrorReset := FALSE;
				State := IDLE;
			END_IF
		END_IF
END_CASE

(*Updates Index 0 of the Drive Message Structure with current drive state info*)
//IF DriveMsgUpdateTimer.Q THEN
//	HARV.DriveLog.AddMsg(TimeStamp 			:= HARV.TimeTracker.TimeStamp,
//						LeftVelocity 		:= DriveLeft.PD6_IN.ActualVelocity,
//						LeftSteeringAngle 	:= LeftWheelAngleActual,
//						RightSteeringAngle 	:= RightWheelAngleActual,
//						LeftCurrent 		:= DriveLeft.PD6_IN.ActiveCurrent,
//						LeftStatusCode 		:= DriveLeft.PD6_IN.StatusWord,
//						RightVelocity 		:= DriveRight.PD6_IN.ActualVelocity,
//						RightCurrent 		:= DriveRight.PD6_IN.ActiveCurrent,
//						RightStatusCode 	:= DriveRight.PD6_IN.StatusWord);
//	DriveMsgUpdateTimer.IN := FALSE;
//ELSE
//	DriveMsgUpdateTimer.IN := TRUE;
//END_IF

(*Read actual drive velocities from the SEVCONS in mm/s*)
LeftVelActual := DriveLeft.SEVCON_IN.ActualVelocity;
RightVelActual := DriveRight.SEVCON_IN.ActualVelocity;

(*Read actual wheel positions and calculate actual wheel angles in degrees from steering motors*)
LeftWheelAngleActual := SteerLeft.PD4_IN.ActualPosition;	// Need to convert to degrees
RightWheelAngleActual := SteerRight.PD4_IN.ActualPosition;	// Need to convery to degrees

TimeInState := TimeInState + T#2MS;
//DriveMsgUpdateTimer();
DriveLeft(SEVCON_IN := DriveLeftIN);
DriveRight(SEVCON_IN := DriveRightIN);
SteerLeft(PD4_IN := SteerLeftIN);
SteerRight(PD4_IN := SteerRightIN);

METHOD CalcDiffVelocity : BOOL
VAR_INPUT
	DriveVelInput	: LREAL;
END_VAR
IF SteeringAngleInput <> 0 THEN
	LeftVelCommand := DriveVelInput * (ICC_R + (CONFIG.RearTrackWidth / 2)) / ICC_R;
	RightVelCommand := DriveVelInput * (ICC_R - (CONFIG.RearTrackWidth / 2)) / ICC_R;
ELSE
	LeftVelCommand := DriveVelInput;
	RightVelCommand := DriveVelInput;
END_IF
END_METHOD

METHOD CalcWheelAngle : BOOL
VAR_INPUT
	SteeringAngleInput	: LREAL;		// degrees
END_VAR
VAR
	RightWheelCenterAngle	: LREAL;
	RightSteerCenterAngle	: LREAL;
	LeftWheelCenterAngle	: LREAL;
	LeftSteerCenterAngle	: LREAL;
	EffectiveWheelBase		: REAL;
END_VAR
EffectiveWheelBase := CONFIG.WheelBase + CONFIG.CasterOffset;

IF SteeringAngleInput > MaxSteeringAngle THEN
	ICC_R := CONFIG.WheelBase / TAN(DEG_TO_RAD(MaxSteeringAngle));
ELSIF SteeringAngleInput < -MaxSteeringAngle THEN
	ICC_R := CONFIG.WheelBase / TAN(DEG_TO_RAD(-MaxSteeringAngle));
ELSE
	ICC_R := CONFIG.WheelBase / TAN(DEG_TO_RAD(SteeringAngleInput));		// Calculate radius of curvature relative to the ICC
END_IF

RightWheelCenterAngle := RAD_TO_DEG(ATAN(EffectiveWheelBase/(ICC_R - (CONFIG.FrontTrackWidth / 2)))); 
LeftWheelCenterAngle := RAD_TO_DEG(ATAN(EffectiveWheelBase/(ICC_R + (CONFIG.FrontTrackWidth / 2))));

RightSteerCenterAngle := RAD_TO_DEG(ASIN((CONFIG.CasterOffset)/(SQRT(EXPT((ICC_R - (CONFIG.FrontTrackWidth / 2)),2) + EXPT(EffectiveWheelBase,2)))));
LeftSteerCenterAngle := RAD_TO_DEG(ASIN((CONFIG.CasterOffset)/(SQRT(EXPT((ICC_R + (CONFIG.FrontTrackWidth / 2)),2) + EXPT(EffectiveWheelBase,2)))));

IF SteeringAngleInput < 0 THEN
	RightWheelAngleCommand := RightWheelCenterAngle + RightSteerCenterAngle;
	LeftWheelAngleCommand := LeftWheelCenterAngle + LeftSteerCenterAngle;
ELSE
	RightWheelAngleCommand := RightWheelCenterAngle - RightSteerCenterAngle;
	LeftWheelAngleCommand := LeftWheelCenterAngle - LeftSteerCenterAngle;
END_IF

SteerLeftAngleTest := LeftWheelAngleCommand;
SteerRightAngleTest	:= RightWheelAngleCommand;

//RightWheelAngle := RAD_TO_DEG(ATAN(CONFIG.WheelBase/(ICC_R - (CONFIG.FrontTrackWidth / 2))));
//LeftWheelAngle := RAD_TO_DEG(ATAN(CONFIG.WheelBase/(ICC_R + (CONFIG.FrontTrackWidth / 2))));
END_METHOD

METHOD ReadButton : BOOL
VAR
	SwitchThreshold	: INT := 1000;
	LowThreshold 	: INT := 500;
END_VAR
IF JoyStick_Button > SwitchThreshold THEN
	ManualDriveEnable := FALSE;
ELSIF JoyStick_Button < SwitchThreshold AND JoyStick_Button > LowThreshold THEN
	ManualDriveEnable := TRUE;
ELSE
	//ManualDriveEnable := FALSE;
END_IF
END_METHOD

END_FUNCTION_BLOCK

// ---- POUs/Device Level Function Blocks/FB_SEVCON.TcPOU
FUNCTION_BLOCK FB_SEVCON
VAR_INPUT
	SEVCON_IN 		: ST_SEVCON_IN;
	Enable			: BOOL;
	ErrorReset		: BOOL;
	TargetVelocity	: UDINT;
	Self			: INT;
END_VAR
VAR_OUTPUT
	SEVCON_OUT : ST_SEVCON_OUT;
	Error		: BOOL;
	ErrorCode	: INT;
	Ready		: BOOL;
	Running		: BOOL;
END_VAR
VAR
	State		: (DEFAULT, INIT, SWITCH_ON_DISABLED, READY_TO_SWITCH_ON, SWITCHED_ON, OPERATION_ENABLED, ERROR);
	PrevState 	: (DEFAULT, INIT, SWITCH_ON_DISABLED, READY_TO_SWITCH_ON, SWITCHED_ON, OPERATION_ENABLED, ERROR);
	TimeInState	: TIME;
	StateEntry 	: BOOL;
	SwitchOn	: BOOL;
	SDO_Write		: FB_SDO_WRITE;
	SDO_WriteData	: ARRAY[0..255] OF BYTE;
	SDO_Read		: FB_SDO_READ;
	SDO_ReadData	: ARRAY[0..255] OF BYTE;
	PreChargeTimer	: TON;
	PreChargeDelay	: TIME := T#3S;
	PreChargeActive	: BOOL;
	
	HiSpeedKp		: BYTE;
	HiSpeedKi		: BYTE;
	LoSpeedKp		: BYTE;
	LoSpeedKi		: BYTE;
END_VAR
VAR CONSTANT
	VoltageMult		: REAL := 0.0625;	// Multiply by voltage params for actual voltages
	MinCapVoltage	: REAL := 40.0;		// check w/ Cedric
END_VAR



IF State <> PrevState THEN
	StateEntry := TRUE;
	PrevState := State;
ELSE
	StateEntry := FALSE;
END_IF

CASE State OF
	DEFAULT:
		State := INIT;
		
	INIT:
		// Set initial parameters
		
		Ready := FALSE;
		SEVCON_OUT.ControlWord := SevConControlWord.DisableVoltage;
		PreChargeTimer.PT := PreChargeDelay;
		
		State := SWITCH_ON_DISABLED;
		
		
	SWITCH_ON_DISABLED:
		IF StateEntry THEN
			SEVCON_OUT.ControlWord := SevConControlWord.DisableVoltage;
			SEVCON_OUT.TargetVelocity := 0;
			SEVCON_OUT.ContactorOutput := 0;
			SEVCON_OUT.BrakeOutput := 0;
		END_IF
		
		IF (SEVCON_IN.StatusWord AND SevConStatusWord.SwitchOnDisabled) = SevConStatusWord.SwitchOnDisabled THEN
			SEVCON_OUT.ControlWord := SevConControlWord.Shutdown;
			State := READY_TO_SWITCH_ON;
		END_IF
		
	READY_TO_SWITCH_ON:
		IF StateEntry THEN
			IF (SEVCON_IN.CapacitorVoltage * VoltageMult) < MinCapVoltage THEN
				PreCharge(TRUE);
			END_IF
			PreChargeTimer.IN := TRUE;
		END_IF
		
		IF ((SEVCON_IN.CapacitorVoltage * VoltageMult) > MinCapVoltage) AND PreChargeTimer.Q THEN
			SEVCON_OUT.ContactorOutput := 65535;
			PreCharge(FALSE);
			SwitchOn := TRUE;
			PreChargeTimer.IN := FALSE;
		END_IF
		
		IF SwitchOn AND ((SEVCON_IN.StatusWord AND SevConStatusWord.ReadyToSwitchon) = SevConStatusWord.ReadyToSwitchon) THEN
			SEVCON_OUT.ControlWord := SevConControlWord.SwitchOn;
			State := SWITCHED_ON;
		END_IF
	
	SWITCHED_ON:
		IF StateEntry THEN
			//
		END_IF
		
		IF (SEVCON_IN.StatusWord AND SevConStatusWord.Switchedon) = SevConStatusWord.Switchedon THEN
			Ready := TRUE;
		ELSE
			Ready := FALSE;
		END_IF
		
		IF Enable AND Ready THEN
			SEVCON_OUT.ControlWord := SevConControlWord.EnableOperation;
			State := OPERATION_ENABLED;
		END_IF

	OPERATION_ENABLED:
		IF StateEntry THEN
			SEVCON_OUT.BrakeOutput := 65535;
			Running := TRUE;
		END_IF
		
		IF NOT Enable THEN
			Running := FALSE;
			SEVCON_OUT.TargetVelocity := 0;
			IF SEVCON_IN.ActualVelocity = 0 THEN
				SEVCON_OUT.BrakeOutput := 0;
				SEVCON_OUT.ControlWord := SevConControlWord.DisableOperation;
				State := SWITCHED_ON;
			END_IF
		ELSE
			SEVCON_OUT.TargetVelocity := TargetVelocity;
		END_IF
	
	ERROR:
		IF StateEntry THEN
			Ready := FALSE;
			Error := TRUE;
		END_IF
		
		IF ErrorReset THEN
			SEVCON_OUT.ControlWord := SevConControlWord.FaultReset;
			IF (SEVCON_IN.StatusWord AND SevConStatusWord.Fault) = 0 THEN
				Error := FALSE;
				ErrorReset := FALSE;
				State := SWITCH_ON_DISABLED;
			END_IF
		END_IF
END_CASE

IF (SEVCON_IN.StatusWord AND SevConStatusWord.Fault) = SevConStatusWord.Fault THEN
	State := ERROR;
END_IF

PreChargeTimer();

METHOD PreCharge : BOOL
VAR_INPUT
	Start	: BOOL;
END_VAR
IF Start THEN
	SDO_WriteData[0] := 16#1;
	PreChargeActive := TRUE;
ELSIF NOT Start THEN
	SDO_WriteData[0] := 16#0;
	PreChargeActive := FALSE;
END_IF

SDO_WRITE(ADSNetID := '5.117.40.235.3.1',
		PortNr := CONFIG.SevCon_Port[self-1],
		CO_Index := INDEX.PreChargeActivate,
		CO_SubIndex := 0,
		DataLength := 1,
		StartWriting := TRUE,
		WriteData := SDO_WriteData);
END_METHOD

METHOD WriteTuningValues : BOOL
VAR_INPUT
	KpHi	: BYTE;
	KiHi	: BYTE;
	KpLo	: BYTE;
	KiLo	: BYTE;
END_VAR
END_METHOD

END_FUNCTION_BLOCK

// ---- POUs/Device Level Function Blocks/FB_SDO_WRITE.TcPOU
FUNCTION_BLOCK FB_SDO_WRITE
VAR_INPUT
	ADSNetID		: STRING(23);   			(* The AMSNetID addresses the EL6751. Can be empty if only one local single channel card is present*)
    PortNr			: WORD;           			(* The Port No. addresses the CANopen Node (see System Manager) *)
    CO_Index		: DWORD;        			(* This is the Index of the CANopen Object Dictionary Entry*)
    CO_SubIndex		: DWORD;     				(*This is the Sub-Index of the CANopen Object Dictionary Entry*)
    DataLength		: DWORD;      				(* This is the Length of the CANopen Object Dictionary Entry*)
    StartWriting	: BOOL;     				(*only reset to FALSE after WriteDataFinished=TRUE*)
    WriteData		: ARRAY[0..255] OF BYTE; 	(*This array contains the data to be written to the CANopen Object Dictionary*)
END_VAR
VAR_OUTPUT
	WriteDataFinished	: BOOL;
    Error				: DWORD;
END_VAR
VAR
	state		: BYTE := 0;
    ADSWRITE	: ADSWRITE;
END_VAR

CASE
state OF
    0:
        IF StartWriting THEN
           WriteDataFinished := FALSE;
           Error := 0;
           ADSWrite(
               NETID:= ADSNetID,
               PORT:= PortNr,
               IDXGRP:= CO_Index,
               IDXOFFS:= CO_SubIndex,
               LEN:= DataLength,
               SRCADDR:= ADR(WriteData),
               WRITE:= TRUE,
               TMOUT := T#1s
               );
           IF ADSWrite.err THEN
               state := 2;
               WriteDataFinished := TRUE;
               Error := ADSWrite.ErrId;
           ELSE
               state := 1;
           END_IF
        ELSE
           ADSWrite(
               NETID:= '',
               PORT:= PortNr,
               IDXGRP:= CO_Index,
               IDXOFFS:= CO_SubIndex,
               LEN:= DataLength,
               SRCADDR:= ADR(WriteData),
               WRITE:= FALSE,
               TMOUT := T#1s
               );
        END_IF
    1:
        ADSWrite(WRITE:= FALSE);
        IF ADSWrite.err THEN
           state := 2;
           WriteDataFinished := TRUE;
           Error := ADSWrite.ErrId;
        ELSE
           IF NOT ADSWrite.busy THEN
               state := 2;
               WriteDataFinished := TRUE;
           END_IF
        END_IF
    2:
        ADSWrite(WRITE:= FALSE);
        state := 0;
END_CASE

END_FUNCTION_BLOCK

// ---- POUs/Device Level Function Blocks/FB_SDO_READ.TcPOU
FUNCTION_BLOCK FB_SDO_READ
VAR_INPUT
	ADSNetID:STRING(23); (* The AMSNetID addresses the EL6751. Can be empty if only one local single channel card is present*)
    PortNr:WORD;         (* This Port No. addresses the CANopen Node (see System Manager) *)
    CO_Index:DWORD;      (* This is the Index of the CANopen Object Dictionary Entry*)
    CO_SubIndex:DWORD;   (* This is the Sub-Index of the CANopen Object Dictionary Entry*)
    DataLength:DWORD;    (* This is the Length of the CANopen Object Dictionary Entry*)
    StartReading:BOOL;   (* only reset to FALSE after ReadDataAvailable=TRUE*)
END_VAR
VAR_OUTPUT
	ReadData:ARRAY[0..255] OF BYTE;
    ReadDataAvailable:BOOL;
    Error:DWORD;
END_VAR
VAR
	state:BYTE := 0;
    ADSREAD:ADSREAD;
END_VAR

CASE
state OF
    0:
        IF StartReading THEN
           ReadDataAvailable := FALSE;
           Error := 0;
           ADSRead(
               NETID:= ADSNetID,
               PORT:= PortNr,
               IDXGRP:= CO_Index,
               IDXOFFS:= CO_SubIndex,
               LEN:= DataLength,
               DESTADDR:= ADR(ReadData),
               READ:= TRUE,
               TMOUT := T#1s
               );
           IF ADSRead.err THEN
               state := 2;
               ReadDataAvailable := TRUE;
               Error := ADSRead.ErrId;
           ELSE
               state := 1;
           END_IF
        ELSE
           ADSRead(
               NETID:= ADSNetID,
               PORT:= PortNr,
               IDXGRP:= CO_Index,
               IDXOFFS:= CO_SubIndex,
               LEN:= DataLength,
               DESTADDR:= ADR(ReadData),
               READ:= FALSE,
               TMOUT := T#1s
           );
        END_IF
    1:
        ADSRead(READ:= FALSE);
        IF ADSRead.err THEN
           state := 2;
           ReadDataAvailable := TRUE;
           Error := ADSRead.ErrId;
        ELSE
           IF NOT ADSRead.busy THEN
               state := 2;
               ReadDataAvailable := TRUE;
           END_IF
        END_IF
    2:
        ADSRead(READ:= FALSE);
        state := 0;
END_CASE

END_FUNCTION_BLOCK

// ---- POUs/Device Level Function Blocks/FB_PD4.TcPOU
FUNCTION_BLOCK FB_PD4
VAR_INPUT
	PD4_IN 			: ST_PD4_IN;
	Enable 			: BOOL;
	ErrorReset 		: BOOL;
	TargetVelocity 	: INT;
	TargetPosition	: DINT;			// Check variable type
	Self 			: INT;
END_VAR
VAR_OUTPUT
	PD4_OUT : ST_PD4_OUT;
	Ready 	: BOOL;
	Error	: BOOL;
END_VAR
VAR
//	State 		: DINT;
	State		: (DEFAULT, INIT, SWITCH_ON_DISABLED, READY_TO_SWITCH_ON, SWITCHED_ON, OPERATION_ENABLED, ERROR);
	PrevState 	: (DEFAULT, INIT, SWITCH_ON_DISABLED, READY_TO_SWITCH_ON, SWITCHED_ON, OPERATION_ENABLED, ERROR);
	StateEntry 	: BOOL;
	Homed		: BOOL;
END_VAR

// POWER FSM State Machine for EtherCAT PD4 Control

IF State <> PrevState THEN
	StateEntry := TRUE;
	PrevState := State;
ELSE
	StateEntry := FALSE;
END_IF

CASE State OF
	DEFAULT:
		State := INIT;
		
	INIT:
		Ready := FALSE;
		PD4_OUT.ControlWord := PD4ControlWord.PulseInhibit;
		PD4_OUT.Polarity := PD4Polarity.Positive;
		
		PD4_OUT.OperationMode := PD4OperationMode.HomingMode;
		PD4_OUT.HomingMethod := 35;									// Zero at current position
		PD4_OUT.ControlWord := PD4ControlWord.StartHoming;
		
		IF PD4_IN.ActualPosition = 0 THEN
			SetMode(PD4OperationMode.ProfilePositionMode);
			SetAbsoluteMotion();
//			SetMode(PD4OperationMode.VelocityMode);
			State := SWITCH_ON_DISABLED;
		END_IF

	SWITCH_ON_DISABLED:
		IF StateEntry THEN
			PD4_OUT.ControlWord := PD4ControlWord.PulseInhibit;
			PD4_OUT.TargetVelocity := 0;
		END_IF
		
		IF ((PD4_IN.StatusWord AND PD4StatusWord.SwitchOnDisabled) = PD4StatusWord.SwitchOnDisabled) THEN
			PD4_OUT.ControlWord := PD4ControlWord.Shutdown;
			State := READY_TO_SWITCH_ON;
		END_IF
		
	READY_TO_SWITCH_ON:
		IF ((PD4_IN.StatusWord AND PD4StatusWOrd.ReadyToSwitchOn) = PD4StatusWOrd.ReadyToSwitchOn) THEN
			PD4_OUT.ControlWord := PD4ControlWord.SwitchOn;
			State := SWITCHED_ON;
		END_IF
		
	SWITCHED_ON:
		IF StateEntry THEN
			Ready := TRUE;
		END_IF
		
		IF (((PD4_IN.StatusWord AND PD4StatusWOrd.SwitchedOn) = PD4StatusWOrd.SwitchedOn) AND Enable) THEN
			PD4_OUT.TargetPosition := PD4_IN.ActualPosition;
			PD4_OUT.ControlWord := PD4ControlWord.EnableOperation;
			State := OPERATION_ENABLED;
		END_IF
		
	OPERATION_ENABLED:
		IF StateEntry THEN
			PD4_OUT.TargetPosition := PD4_IN.ActualPosition;
			TargetPosition := PD4_IN.ActualPosition;
		END_IF
		
		PD4_OUT.TargetPosition := TargetPosition;
		ToggleMoveBit();
//		PD4_OUT.TargetVelocity := TargetVelocity;	
		
		IF NOT Enable THEN
//			PD4_OUT.TargetVelocity := 0;
			PD4_OUT.TargetPosition := PD4_IN.ActualPosition;
			PD4_OUT.ControlWord := PD4ControlWord.DisableOperation;
			State := SWITCHED_ON;
		END_IF
		
	ERROR:
		IF StateEntry THEN
			Ready := FALSE;
			Error := TRUE;	
		END_IF
		
		IF ErrorReset THEN
			PD4_OUT.ControlWord := PD4ControlWord.FaultReset;
			IF ((PD4_IN.StatusWord AND PD4StatusWOrd.Fault) = 0) THEN
				Error := FALSE;
				State := SWITCH_ON_DISABLED;
			END_IF
		END_IF
END_CASE

IF ((PD4_IN.StatusWord AND PD4StatusWord.Fault) = PD4StatusWord.Fault) THEN
	State := ERROR;
END_IF

METHOD SetAbsoluteMotion : BOOL
VAR_INPUT
END_VAR
PD4_OUT.ControlWord := PD4_OUT.ControlWord OR PD4ControlWord.AbsoluteMotion;
END_METHOD

METHOD SetMaxCurrent : BOOL
VAR_INPUT
END_VAR
END_METHOD

METHOD SetMode : BOOL
VAR_INPUT
	OperationMode	: PD4OperationMode;
END_VAR
PD4_OUT.OperationMode := OperationMode;
PD4_OUT.SubmodeSelect := 1;
END_METHOD

METHOD SetMotionProfile : BOOL
VAR_INPUT
	Velocity 	: UDINT;
	Accel 		: UDINT;
	Decel 		: UDINT;
END_VAR
PD4_OUT.ProfileVelocity := Velocity;
PD4_OUT.Accel := Accel;
PD4_OUT.Decel := Decel;
END_METHOD

METHOD ToggleMoveBit : BOOL
VAR_INPUT
END_VAR
IF (PD4_OUT.ControlWord AND PD4ControlWord.StartMove) = PD4ControlWord.StartMove THEN
	PD4_OUT.ControlWord := (PD4_OUT.ControlWord AND (NOT PD4ControlWord.StartMove));
ELSE
	PD4_OUT.ControlWord := (PD4_OUT.ControlWord OR PD4ControlWord.StartMove);
END_IF
END_METHOD

END_FUNCTION_BLOCK

// ---- POUs/Log Level Function Blocks/FB_ERROR_MSG_LOG.TcPOU
FUNCTION_BLOCK FB_ERROR_MSG_LOG
VAR
	Buffer 	: ARRAY[0..MaxBufferSize] OF ST_ERROR_MSG;
	Index	: INT;
END_VAR
VAR CONSTANT
	MaxBufferSize	: INT := 1000;
END_VAR

METHOD AddMsg : BOOL
VAR_INPUT
	TimeStamp	: DT;
	Location	: STRING;
	ErrorCode	: INT;
	Description	: STRING;
END_VAR
VAR
	i	: INT;
END_VAR
FOR i := 0 TO MaxBufferSize DO
	IF Buffer[MaxBufferSize - i].Location = '' THEN
		CONTINUE;
	ELSE
		Buffer[MaxBufferSize - i + 1].Location 		:= Buffer[MaxBufferSize - i].Location;
		Buffer[MaxBufferSize - i + 1].TimeStamp 	:= Buffer[MaxBufferSize - i].TimeStamp;
		Buffer[MaxBufferSize - i + 1].ErrorCode 	:= Buffer[MaxBufferSize - i].ErrorCode;
		Buffer[MaxBufferSize - i + 1].Description 	:= Buffer[MaxBufferSize - i].Description;
	END_IF
END_FOR

Buffer[0].Location 		:= Location;
Buffer[0].Timestamp 	:= TimeStamp;
Buffer[0].ErrorCode 	:= ErrorCode;
Buffer[0].Description 	:= Description;

Index := Index + 1;
END_METHOD

END_FUNCTION_BLOCK

// ---- POUs/Log Level Function Blocks/FB_DRIVE_MSG_LOG.TcPOU
FUNCTION_BLOCK FB_DRIVE_MSG_LOG
VAR
	Buffer	: ARRAY[0..MaxBufferSize] OF ST_DRIVE_MSG;
	Index : INT;
END_VAR
VAR CONSTANT
	MaxBufferSize	: INT := 1000;
END_VAR

METHOD AddMsg : BOOL
VAR_INPUT
	TimeStamp			: DT;
	LeftVelocity		: INT;
	RightVelocity		: INT;
	LeftSteeringAngle	: LREAL;
	RightSteeringAngle	: LREAL;
	LeftCurrent			: REAL;
	RightCurrent		: REAL;
	LeftStatusCode		: UINT;
	RightStatusCode		: UINT;
END_VAR
VAR
	i: INT;
END_VAR
FOR i := 0 TO MaxBufferSize DO
	IF Buffer[MaxBufferSize - i].LeftVelocity = 0.0 THEN
		CONTINUE;
	ELSE
		Buffer[MaxBufferSize - i + 1].TimeStamp 			:= Buffer[MaxBufferSize - i].TimeStamp;
		Buffer[MaxBufferSize - i + 1].LeftVelocity 			:= Buffer[MaxBufferSize - i].LeftVelocity;
		Buffer[MaxBufferSize - i + 1].RightVelocity 		:= Buffer[MaxBufferSize - i].RightVelocity;
		Buffer[MaxBufferSize - i + 1].LeftSteeringAngle 	:= Buffer[MaxBufferSize - i].LeftSteeringAngle;
		Buffer[MaxBufferSize - i + 1].RightSteeringAngle 	:= Buffer[MaxBufferSize - i].RightSteeringAngle;
		Buffer[MaxBufferSize - i + 1].LeftCurrent 			:= Buffer[MaxBufferSize - i].LeftCurrent;
		Buffer[MaxBufferSize - i + 1].RightCurrent 			:= Buffer[MaxBufferSize - i].RightCurrent;
		Buffer[MaxBufferSize - i + 1].LeftStatusCode 		:= Buffer[MaxBufferSize - i].LeftStatusCode;
		Buffer[MaxBufferSize - i + 1].RightStatusCode 		:= Buffer[MaxBufferSize - i].RightStatusCode;
	END_IF
END_FOR

Buffer[0].Timestamp 			:= TimeStamp;
Buffer[0].LeftVelocity 			:= LeftVelocity;
Buffer[0].RightVelocity 		:= RightVelocity;
Buffer[0].LeftSteeringAngle 	:= LeftSteeringAngle;
Buffer[0].RightSteeringAngle 	:= RightSteeringAngle;
Buffer[0].LeftCurrent 			:= LeftCurrent;
Buffer[0].RightCurrent 			:= RightCurrent;
Buffer[0].LeftStatusCode 		:= LeftStatusCode;
Buffer[0].RightStatusCode 		:= RightStatusCode;

Index := Index + 1;
END_METHOD

END_FUNCTION_BLOCK

// ---- POUs/Log Level Function Blocks/FB_TIMETRACKER.TcPOU
FUNCTION_BLOCK FB_TIMETRACKER
VAR_INPUT
END_VAR
VAR_OUTPUT
	TimeStamp		: DT;
END_VAR
VAR
	GetSystemTime	: FB_LOCALSYSTEMTIME;
	TimeStampStruct	: TIMESTRUCT;
END_VAR

GetSystemTime(sNetID := '', bEnable := TRUE, systemTime => TimeStampStruct);
TimeStamp := SYSTEMTIME_TO_DT(TimeStampStruct);

END_FUNCTION_BLOCK

// ---- POUs/SubSystem Level Function Blocks/FB_TILT.TcPOU
FUNCTION_BLOCK FB_TILT
VAR_INPUT
	IMU_Roll				: INT;
	IMU_Pitch				: INT;
	AutoTiltControlEnable	: BOOL;
	ManualTiltControlEnable : BOOL;
	StartupEnable			: BOOL;
	TestModeEnable			: BOOL;
	PressureSwitch			: BOOL;
END_VAR
VAR_OUTPUT
	RollValveLeft	: FB_HYDRAULIC_VALVE;
	RollValveRight	: FB_HYDRAULIC_VALVE;
	PitchValve		: FB_HYDRAULIC_VALVE;
	PumpContactor	: BOOL;
	Error			: BOOL;
	ErrorCode		: DINT;
	Ready			: BOOL;
END_VAR
VAR
	TiltDisplacement		: REAL;
	TiltLeftDisplacement	: REAL;
	TiltRightDisplacement	: REAL;
	
	RollAngle				: REAL;
	PitchAngle				: REAL;
	SlopeAngle				: REAL;
	
	State					: (DEFAULT, INIT, IDLE, STARTUP, MANUAL, AUTO, TEST, ERROR);
	PrevState				: (DEFAULT, INIT, IDLE, STARTUP, MANUAL, AUTO, TEST, ERROR);
	StateEntry				: BOOL;
	
	StartHoming				: BOOL;
	Homed					: BOOL;
	CurrentAxis				: INT;
	RearStartPosition		: BOOL;
	FrontStartPosition		: BOOL;
	InStartPosition			: BOOL;
	StartupTimer			: TON;
	StartDelay				: TIME := T#1500MS;
	PumpStartupTimer		: TON;
	PumpStartupDelay		: TIME := T#2000MS;
	CylinderBumpTimer		: TON;
	CylinderBumpDelay		: TIME := T#300MS;
	
	RollAxisLevel			: BOOL;
	PitchAxisLevel			: BOOL;
	
	RollCW_Command			: BOOL;
	RollCCW_Command			: BOOL;
	PitchUp_Command			: BOOL;
	PitchDown_Command		: BOOL;
	Raise_Command			: BOOL;
	Lower_Command			: BOOL;
	Level_Command			: BOOL;
	
	IMU_Roll_Avg			: INT;
	RollDataBuffer			: ARRAY[0..9] OF INT;
	IMU_Pitch_Avg			: INT;
	PitchDataBuffer			: ARRAY[0..9] OF INT;
	
	PressureSwitch_FTRIG	: F_TRIG;
	RearLeftCheck			: BOOL;
	RearRightCheck			: BOOL;
	FrontCheck				: BOOL;
	PitchAngleStart			: REAL;
	RollAngleStart			: REAL;
END_VAR
VAR CONSTANT
	IMU_DeadBand			: INT := 400;
	IMU_Center				: INT := 16535;
	IMU_MaxAngle			: REAL := 30;
	RollControlThreshold	: REAL := 1.0;		// angular delta where the tilt controller kicks in
	PitchControlThreshold	: REAL := 1.0;
	PitchStartupAngle		: REAL := 7.0;		// roughly half stroke on rear cylinders when starting flat
	MaxRollAngle			: REAL := 10;
	MaxPitchAngle			: REAL := 20;
END_VAR



IF State <> PrevState THEN
	StateEntry := TRUE;
	PrevState := State;
ELSE
	StateEntry := FALSE;
END_IF

PressureSwitch_FTRIG.CLK := PressureSwitch;

CASE State OF
	DEFAULT:
		State := INIT;
		
	INIT:
		IF StateEntry THEN
			RearStartPosition := FALSE;
			FrontStartPosition := FALSE;
			InStartPosition := FALSE;
			StartupTimer.PT := StartDelay;
			PumpStartupTimer.PT := PumpStartupDelay;
			CylinderBumpTimer.PT := CylinderBumpDelay;
		END_IF
		
		State := IDLE;
		
	IDLE:
		IF StateEntry THEN
			Hold(TRUE);
		END_IF
		
		IF AutoTiltControlEnable AND InStartPosition THEN
			State := Auto;
		ELSIF ManualTiltControlEnable THEN
			State := MANUAL;
		ELSIF StartupEnable THEN
			State := STARTUP;
		ELSIF TestModeEnable THEN
			State := TEST;
		END_IF
	
	STARTUP:
		IF StateEntry THEN
			PumpContactor := TRUE;
			PumpStartupTimer.IN := TRUE;
			PitchAngleStart := PitchAngle;
			RollAngleStart	:= RollAngle;
		END_IF	
		
		IF PumpStartupTimer.Q THEN
			IF (NOT RearStartPosition) AND (NOT FrontStartPosition) THEN
				RollValveLeft.Extend();
				RollValveRight.Extend();
				IF PitchAngle <= (PitchAngleStart - PitchStartupAngle) THEN
					RollValveLeft.Neutral();
					RolLValveRight.Neutral();
					StartupTimer.IN := FALSE;
					RearStartPosition := TRUE;
				END_IF
			ELSIF( RearStartPosition) AND (NOT FrontStartPosition) THEN
				PitchUp(TRUE);
				IF PitchAngle >= PitchAngleStart THEN
					PitchUp(FALSE);
					FrontStartPosition := TRUE;
					InStartPosition := TRUE;
				END_IF
			END_IF
		END_IF
		
		IF NOT StartupEnable OR InStartPosition THEN
			PumpStartupTimer.IN := FALSE;
			Hold(TRUE);
			PumpContactor := FALSE;
			StartupEnable := FALSE;
			State := IDLE;
		END_IF
	
	MANUAL:	
		IF StateEntry THEN
			PumpContactor := TRUE;
		END_IF
		
		IF RollCW_Command THEN
			RollCW(TRUE);
			IF RollAngle >= 8.0 THEN
				RollCW(FALSE);
				RollCW_Command := FALSE;
			END_IF
		ELSIF RollCCW_Command THEN
			RollCCW(TRUE);
			IF RollAngle <= -8.0 THEN
				RollCCW(FALSE);
				RollCCW_Command := FALSE;
			END_IF
		ELSIF Level_Command THEN
			IF RollAngle > 0 AND NOT RollAxisLevel THEN
				RollCCW(TRUE);
				RollAxisLevel := FALSE;
			ELSIF RollAngle < 0 AND NOT RollAxisLevel THEN
				RollCW(TRUE);
				RollAxisLevel := FALSE;
			ELSE
				RollCW(FALSE);
				RollCCW(FALSE);
				RollAxisLevel := TRUE;
			END_IF
			
			IF PitchAngle > 0 AND RollAxisLevel THEN
				PitchDown(TRUE);
			ELSIF PitchANgle < 0 AND RollAxisLevel THEN
				PitchUp(TRUE);
			ELSE
				PitchValve.Neutral();
				PitchAxisLevel := TRUE;
			END_IF
			
			IF RollAxisLevel AND PitchAxisLevel THEN
				Level_Command := FALSE;
			END_IF
		ELSIF Raise_Command THEN
			Raise(TRUE);
		ELSIF Lower_Command THEN
			Lower(TRUE);
		ELSIF PitchUp_Command THEN
			PitchUp(TRUE);
		ELSIF PitchDown_Command THEN
			PitchDown(TRUE);
		END_IF
		
//		IF PressureSwitch_FTRIG.Q THEN
//			Hold(TRUE);
//			RollCw_Command := FALSE;
//			RollCCW_Command := FALSE;
//			Raise_Command := FALSE;
//			Lower_Command := FALSE;
//			PitchUp_Command := FALSE;
//			PitchDown_Command := FALSE;
//			PumpContactor := FALSE;
//		END_IF
		
		IF NOT ManualTiltControlEnable THEN
			Hold(TRUE);
			PumpContactor := FALSE;
			State := IDLE;
		END_IF
	
	AUTO:
		IF StateEntry THEN
			RollAxisLevel := FALSE;
			PitchAxisLevel := FALSE;
			Hold(TRUE);
		END_IF
		
		IF NOT RollAxisLevel AND NOT PitchAxisLevel THEN
			IF (RollAngle > RollControlThreshold) THEN
				PumpContactor := TRUE;
				IF CylinderBumpTimer.Q THEN
					CylinderBumpTimer.IN := FALSE;
					IF NOT RollValveLeft.SolenoidRetract AND NOT RollValveRight.SolenoidExtend THEN
						RollValveLeft.Retract();
					ELSIF RollValveLeft.SolenoidRetract THEN
						RollValveLeft.Neutral();
						RollValveRight.Extend();
					ELSIF RollValveRight.SolenoidExtend THEN
						RollValveLeft.Retract();
						RollValveRight.Neutral();
					END_IF
				ELSE
					CylinderBumpTimer.IN := TRUE;
				END_IF
				//RollCCW(TRUE);
			ELSIF RollAngle < -RollControlThreshold THEN
				PumpContactor := TRUE;
				IF CylinderBumpTimer.Q THEN
					CylinderBumpTimer.IN := FALSE;
					IF NOT RollValveLeft.SolenoidExtend AND NOT RollValveRight.SolenoidRetract THEN
						RollValveLeft.Extend();
					ELSIF RollValveLeft.SolenoidExtend THEN
						RollValveLeft.Neutral();
						RollValveRight.Retract();
					ELSIF RollValveRight.SolenoidRetract THEN
						RollValveLeft.Extend();
						RollValveRight.Neutral();
					END_IF
				ELSE
					CylinderBumpTimer.IN := TRUE;
				END_IF
				//RollCW(TRUE);
			ELSIF RollAngle > -RollControlThreshold AND RollAngle < RollControlThreshold THEN
				RollAxisLevel := TRUE;
				RollCCW(FALSE);
				RollCW(FALSE);
			END_IF
		ELSIF RollAxisLevel AND NOT PitchAxisLevel THEN
			IF PitchAngle > PitchControlThreshold THEN
				PitchDown(TRUE);
			ELSIF PitchAngle < -PitchControlThreshold THEN
				PitchUp(TRUE);
			ELSIF PitchAngle > -PitchControlThreshold AND PitchAngle < PitchControlThreshold THEN
				PitchAxisLevel := TRUE;
				PitchDown(FALSE);
				PitchUp(FALSE);
			END_IF
		END_IF
		
//		IF PressureSwitch_FTRIG.Q THEN
//			Hold(TRUE);
//			PumpStartupTimer.IN := FALSE;
//		END_IF
		
		(*From the slope angle, calculate the required actuator displacement for leveling*)
		CalcDisplacement(RollAngle);
		
		IF NOT AutoTiltControlEnable OR (PitchAxisLevel AND RollAxisLevel) THEN
			PumpStartupTimer.IN := FALSE;
			Hold(TRUE);
			PumpContactor := FALSE;
			AutoTiltControlEnable := FALSE;
			State := IDLE;
		END_IF
	
	TEST:
		IF StateEntry THEN
			Homed := FALSE;
			CurrentAxis := 1;
			PumpContactor := TRUE;
		END_IF
		
		IF StartHoming THEN
			IF CurrentAxis = 1 THEN
				RollValveLeft.Extend();
				IF PressureSwitch_FTRIG.Q THEN
					RollValveLeft.Neutral();
					CurrentAxis := 2;
				END_IF
			ELSIF CurrentAxis = 2 THEN
				RollValveRight.Extend();
				IF PressureSwitch_FTRIG.Q THEN
					RollValveRight.Neutral();
					CurrentAxis := 3;
				END_IF
			ELSIF CurrentAxis = 3 THEN
				PitchValve.Extend();
				IF PressureSwitch_FTRIG.Q THEN
					PitchValve.Neutral();
					CurrentAxis := 0;
				END_IF
			ELSIF CurrentAxis = 0 THEN
				Lower(TRUE);
				IF PressureSwitch_FTRIG.Q THEN
					Hold(TRUE);
					Homed := TRUE;
					StartHoming := FALSE;
				END_IF
			END_IF
		END_IF
		
		IF NOT TestModeEnable THEN
			Hold(TRUE);
			PumpContactor := FALSE;
			State := IDLE;
		END_IF
		
	ERROR:
		IF StateEntry THEN
			//
		END_IF
END_CASE

(*Calculates a moving average of the last 10 data points (20ms) for use in the angle calculation*)
MovingAverage(IMU_Roll, IMU_Pitch);

(*Read input from the IMU in the roll direction and calculate the slope angle*)
IF IMU_Roll_Avg > (IMU_Center + IMU_DeadBand) THEN
	RollAngle := INT_TO_REAL(IMU_Roll_Avg - (IMU_Center + IMU_DeadBand)) / (IMU_Center - IMU_DeadBand) * IMU_MaxAngle;
ELSIF IMU_Roll_Avg < (IMU_Center - IMU_DeadBand) THEN
	RollAngle := INT_TO_REAL(IMU_Roll_Avg - (IMU_Center - IMU_DeadBand)) / (IMU_Center - IMU_DeadBand) * IMU_MaxAngle;
ELSE
	RollAngle := 0;
END_IF

IF IMU_Pitch_Avg > (IMU_Center + IMU_DeadBand) THEN
	PitchAngle := INT_TO_REAL(IMU_Pitch_Avg - (IMU_Center + IMU_DeadBand)) / (IMU_Center - IMU_DeadBand) * IMU_MaxAngle;
ELSIF IMU_Pitch_Avg < (IMU_Center - IMU_DeadBand) THEN
	PitchAngle := INT_TO_REAL(IMU_Pitch_Avg - (IMU_Center - IMU_DeadBand)) / (IMU_Center - IMU_DeadBand) * IMU_MaxAngle;
ELSE
	PitchAngle := 0;
END_IF

PressureSwitch_FTRIG();
StartupTimer();
PumpStartupTimer();
CylinderBumpTimer();

METHOD CalcDisplacement : BOOL
VAR_INPUT
	RollAngle	: REAL;
END_VAR
TiltDisplacement := ABS((CONFIG.RearTrackWidth) * SIN(DEG_TO_RAD(RollAngle)));

//TiltRightDisplacement := (CONFIG.RearTrackWidth / 2) * SIN(DEG_TO_RAD(SlopeAngle));
//TiltLeftDisplacement := (-CONFIG.RearTrackWidth / 2) * SIN(DEG_TO_RAD(SlopeAngle));

IF RollAngle < 0 THEN
	TiltLeftDisplacement := TiltDisplacement;
	TiltRightDisplacement := 0;
ELSIF RollAngle > 0 THEN
	TiltLeftDisplacement := 0;
	TiltRightDisplacement := TiltDisplacement;
ELSE
	TiltLeftDisplacement := 0;
	TiltRightDisplacement := 0;
END_IF
END_METHOD

METHOD CheckValveState : BOOL
VAR_INPUT
END_VAR
END_METHOD

METHOD Hold : BOOL
VAR_INPUT
	Run	: BOOL;
END_VAR
IF Run THEN
	RollValveLeft.Neutral();
	RollValveRight.Neutral();
	PitchValve.Neutral();
ELSE
	//
END_IF
END_METHOD

METHOD Lower : BOOL
VAR_INPUT
	Run	: BOOL;
END_VAR
IF Run THEN
	RollValveLeft.Retract();
	RollValveRight.Retract();
	PitchValve.Retract();
ELSE
	RollValveLeft.Neutral();
	RollValveRight.Neutral();
	PitchValve.Neutral();
END_IF
END_METHOD

METHOD MovingAverage : INT
VAR_INPUT
	IMU_Roll_Input	: INT;
	IMU_Pitch_Input	: INT;
END_VAR
VAR
	ArraySumRoll	: DINT := 0;
	ArraySumPitch	: DINT := 0;
	i	: INT;
END_VAR
FOR i := 0 TO 8 DO
	//ArraySumRoll := ArraySumRoll + RollDataBuffer[i];
	//ArraySumPitch := ArraySumPitch + PitchDataBuffer[i];
	RollDataBuffer[i + 1] := RollDataBuffer[i];
	PitchDataBuffer[i + 1] := PitchdataBuffer[i];
END_FOR

RollDataBuffer[0] := IMU_Roll_Input;
PitchDataBuffer[0] := IMU_Pitch_Input;

ArraySumRoll := RollDataBuffer[0] + RollDataBuffer[1] + RollDataBuffer[2] + RollDataBuffer[3] +
				RollDataBuffer[4] + RollDataBuffer[5] + RollDataBuffer[6] + RollDataBuffer[7] +
				RollDataBuffer[8] + RollDataBuffer[9];
				
ArraySumPitch := PitchDataBuffer[0] + PitchDataBuffer[1] + PitchDataBuffer[2] + PitchDataBuffer[3] +
				PitchDataBuffer[4] + PitchDataBuffer[5] + PitchDataBuffer[6] + PitchDataBuffer[7] +
				PitchDataBuffer[8] + PitchDataBuffer[9];

IMU_Roll_Avg := REAL_TO_INT(ArraySumRoll / 10);
IMU_Pitch_Avg := REAL_TO_INT(ArraySumPitch / 10);
END_METHOD

METHOD PitchDown : BOOL
VAR_INPUT
	Run	: BOOL;
END_VAR
IF Run THEN
	PitchValve.Retract();
ELSE
	PitchValve.Neutral();
END_IF
END_METHOD

METHOD PitchUp : BOOL
VAR_INPUT
	Run	: BOOL;
END_VAR
IF Run THEN
	PitchValve.Extend();
ELSE
	PitchValve.Neutral();
END_IF
END_METHOD

METHOD Raise : BOOL
VAR_INPUT
	Run	: BOOL;
END_VAR
IF Run THEN
	RollValveLeft.Extend();
	RollValveRight.Extend();
	PitchValve.Extend();
ELSE
	RollValveLeft.Neutral();
	RollValveRight.Neutral();
	PitchValve.Neutral();
END_IF
END_METHOD

METHOD RollCCW : BOOL
VAR_INPUT
	Run	: BOOL;
END_VAR
IF Run THEN
	RollValveLeft.Retract();
	RollValveRight.Extend();
ELSE
	RollValveLeft.Neutral();
	RollValveRight.Neutral();
END_IF
END_METHOD

METHOD RollCW : BOOL
VAR_INPUT
	Run	: BOOL;
END_VAR
IF Run THEN
	RollValveLeft.Extend();
	RollValveRight.Retract();
ELSE
	RollValveLeft.Neutral();
	RollValveRight.Neutral();
END_IF
END_METHOD

END_FUNCTION_BLOCK

// ---- POUs/Device Level Function Blocks/FB_HYDRAULIC_VALVE.TcPOU
FUNCTION_BLOCK FB_HYDRAULIC_VALVE
VAR_INPUT
END_VAR
VAR_OUTPUT
	SolenoidExtend	: BOOL;
	SolenoidRetract	: BOOL;
END_VAR
VAR
END_VAR

METHOD Extend : BOOL
VAR_INPUT
END_VAR
SolenoidExtend := TRUE;
SolenoidRetract := FALSE;
END_METHOD

METHOD Neutral : BOOL
VAR_INPUT
END_VAR
SolenoidExtend := FALSE;
SolenoidRetract := FALSE;
END_METHOD

METHOD Retract : BOOL
VAR_INPUT
END_VAR
SolenoidExtend := FALSE;
SolenoidRetract := TRUE;
END_METHOD

END_FUNCTION_BLOCK

// ---- POUs/SubSystem Level Function Blocks/FB_BINFILLER.TcPOU
FUNCTION_BLOCK FB_BINFILLER
VAR_INPUT
	UpLeftConveyor_IN		: ST_PD6_IN;
	UpRightConveyor_IN		: ST_PD6_IN;
	DownLeftConveyor_IN		: ST_PD6_IN;
	DownRightConveyor_IN	: ST_PD6_IN;
	Rotary_IN				: ST_PD6_IN;
	AugerLeft_IN			: ST_PD6_IN;
	AugerRight_IN			: ST_PD6_IN;
	Enable	: BOOL;
END_VAR
VAR_OUTPUT
	UpLeftConveyor		: FB_PD6;
	UpRightConveyor		: FB_PD6;
	DownLeftConveyor	: FB_PD6;
	DownRightConveyor	: FB_PD6;
	Rotary				: FB_PD6;
	AugerLeft			: FB_PD6;
	AugerRight			: FB_PD6;
END_VAR
VAR
	State		: (DEFAULT, INIT, IDLE, MANUAL, AUTO, ERROR);
	PrevState	: (DEFAULT, INIT, IDLE, MANUAL, AUTO, ERROR);
	StateEntry 	: BOOL;
END_VAR



IF State <> PrevState THEN
	StateEntry := TRUE;
	PrevState := State;
ELSE
	StateEntry := FALSE;
END_IF

CASE State OF
	DEFAULT:
		//
	INIT:
		//
	IDLE:
		//
	MANUAL:
		//
	AUTO:
		//
	ERROR:
		//
END_CASE

UpLeftConveyor(PD6_IN := UpLeftConveyor_IN);
UpRightConveyor(PD6_IN := UpRightConveyor_IN);
DownLeftConveyor(PD6_IN := DownLeftConveyor_IN);
DownRightConveyor(PD6_IN := DownRightConveyor_IN);
Rotary(PD6_IN := Rotary_IN);
AugerLeft(PD6_IN := AugerLeft_IN);
AugerRight(PD6_IN := AugerRight_IN);

END_FUNCTION_BLOCK

// ---- POUs/Device Level Function Blocks/FB_PD6.TcPOU
FUNCTION_BLOCK FB_PD6
VAR_INPUT
	PD6_IN 			: ST_PD6_IN;
	Enable 			: BOOL;
	ErrorReset 		: BOOL;
	TargetVelocity 	: INT;
	TargetPosition	: DINT;			// Check variable type
	Self 			: INT;
END_VAR
VAR_OUTPUT
	PD6_OUT : ST_PD6_OUT;
	Ready 	: BOOL;
	Error	: BOOL;
END_VAR
VAR
//	State 		: DINT;
	State		: (DEFAULT, INIT, SWITCH_ON_DISABLED, READY_TO_SWITCH_ON, SWITCHED_ON, OPERATION_ENABLED, ERROR);
	PrevState 	: (DEFAULT, INIT, SWITCH_ON_DISABLED, READY_TO_SWITCH_ON, SWITCHED_ON, OPERATION_ENABLED, ERROR);
	StateEntry 	: BOOL;
	Homed		: BOOL;
END_VAR

// POWER FSM State Machine for EtherCAT PD6 Control

IF State <> PrevState THEN
	StateEntry := TRUE;
	PrevState := State;
ELSE
	StateEntry := FALSE;
END_IF

CASE State OF
	DEFAULT:
		State := INIT;
		
	INIT:
		Ready := FALSE;
		PD6_OUT.ControlWord := PD6ControlWord.PulseInhibit;
		PD6_OUT.Polarity := PD6Polarity.Positive;
		
		PD6_OUT.OperationMode := PD6OperationMode.HomingMode;
		PD6_OUT.HomingMethod := 35;									// Zero at current position
		PD6_OUT.ControlWord := PD6ControlWord.StartHoming;
		
		IF PD6_IN.ActualPosition = 0 THEN
//			SetMode(PD6OperationMode.ProfilePositionMode);
//			SetAbsoluteMotion();
			SetMode(PD6OperationMode.VelocityMode);
			State := SWITCH_ON_DISABLED;
		END_IF

	SWITCH_ON_DISABLED:
		IF StateEntry THEN
			PD6_OUT.ControlWord := PD6ControlWord.PulseInhibit;
			PD6_OUT.TargetVelocity := 0;
		END_IF
		
		IF ((PD6_IN.StatusWord AND PD6StatusWord.SwitchOnDisabled) = PD6StatusWord.SwitchOnDisabled) THEN
			PD6_OUT.ControlWord := PD6ControlWord.Shutdown;
			State := READY_TO_SWITCH_ON;
		END_IF
		
	READY_TO_SWITCH_ON:
		IF ((PD6_IN.StatusWord AND PD6StatusWOrd.ReadyToSwitchOn) = PD6StatusWOrd.ReadyToSwitchOn) THEN
			PD6_OUT.ControlWord := PD6ControlWord.SwitchOn;
			State := SWITCHED_ON;
		END_IF
		
	SWITCHED_ON:
		IF StateEntry THEN
			Ready := TRUE;
		END_IF
		
		IF (((PD6_IN.StatusWord AND PD6StatusWOrd.SwitchedOn) = PD6StatusWOrd.SwitchedOn) AND Enable) THEN
			PD6_OUT.TargetPosition := PD6_IN.ActualPosition;
			PD6_OUT.ControlWord := PD6ControlWord.EnableOperation;
			State := OPERATION_ENABLED;
		END_IF
		
	OPERATION_ENABLED:
		IF StateEntry THEN
			PD6_OUT.TargetPosition := PD6_IN.ActualPosition;
			TargetPosition := PD6_IN.ActualPosition;
		END_IF
		
//		PD6_OUT.TargetPosition := TargetPosition;
//		ToggleMoveBit();
		PD6_OUT.TargetVelocity := TargetVelocity;	
		
		IF NOT Enable THEN
			PD6_OUT.TargetVelocity := 0;
//			PD6_OUT.TargetPosition := PD6_IN.ActualPosition;
			PD6_OUT.ControlWord := PD6ControlWord.DisableOperation;
			State := SWITCHED_ON;
		END_IF
		
	ERROR:
		IF StateEntry THEN
			Ready := FALSE;
			Error := TRUE;	
		END_IF
		
		IF ErrorReset THEN
			PD6_OUT.ControlWord := PD6ControlWord.FaultReset;
			IF ((PD6_IN.StatusWord AND PD6StatusWOrd.Fault) = 0) THEN
				Error := FALSE;
				State := SWITCH_ON_DISABLED;
			END_IF
		END_IF
END_CASE

IF ((PD6_IN.StatusWord AND PD6StatusWord.Fault) = PD6StatusWord.Fault) THEN
	State := ERROR;
END_IF

METHOD SetAbsoluteMotion : BOOL
VAR_INPUT
END_VAR
END_METHOD

METHOD SetMaxCurrent : BOOL
VAR_INPUT
END_VAR
END_METHOD

METHOD SetMode : BOOL
VAR_INPUT
	OperationMode	: PD6OperationMode;
END_VAR
PD6_OUT.OperationMode := OperationMode;
PD6_OUT.SubmodeSelect := 1;
END_METHOD

METHOD SetMotionProfile : BOOL
VAR_INPUT
	Velocity	: UDINT;
	Accel		: UDINT;
	Decel		: UDINT;
END_VAR
PD6_OUT.ProfileVelocity := Velocity;
PD6_OUT.Accel := Accel;
PD6_OUT.Decel := Decel;
END_METHOD

METHOD ToggleMoveBit : BOOL
VAR_INPUT
END_VAR
IF (PD6_OUT.ControlWord AND PD6ControlWord.StartMove) = PD6ControlWord.StartMove THEN
	PD6_OUT.ControlWord := (PD6_OUT.ControlWord AND (NOT PD6ControlWord.StartMove));
ELSE
	PD6_OUT.ControlWord := (PD6_OUT.ControlWord OR PD6ControlWord.StartMove);
END_IF
END_METHOD

END_FUNCTION_BLOCK

// ---- POUs/SubSystem Level Function Blocks/FB_BIN_MANAGER.TcPOU
FUNCTION_BLOCK FB_BIN_MANAGER
VAR_INPUT
	Enable	: BOOL;
END_VAR
VAR_OUTPUT
	FrontForkValve	: FB_HYDRAULIC_VALVE;
	RearForkValve	: FB_HYDRAULIC_VALVE;
	GateStop		: BOOL;
	Error			: BOOL;
	Ready			: BOOL;
END_VAR
VAR
	State 		: (DEFAULT, INIT, IDLE, LOAD, UNLOAD, ERROR);
	PrevState	: (DEFAULT, INIT, IDLE, LOAD, UNLOAD, ERROR);
	StateEntry	: BOOL;
END_VAR



IF State <> PrevState THEN
	StateEntry := TRUE;
	PrevState := State;
ELSE
	StateEntry := FALSE;
END_IF

CASE State OF
	DEFAULT:
		//
	INIT:
		//
	IDLE:
		//
	LOAD:
		//
	UNLOAD:
		//
	ERROR:
		//
END_CASE

END_FUNCTION_BLOCK

// ---- POUs/SubSystem Level Function Blocks/FB_CONVEYANCE.TcPOU
FUNCTION_BLOCK FB_CONVEYANCE
VAR_INPUT
END_VAR
VAR_OUTPUT
END_VAR
VAR
END_VAR

END_FUNCTION_BLOCK

// ---- POUs/FB_READ_HW.TcPOU
FUNCTION_BLOCK FB_READ_HW
VAR_INPUT
END_VAR
VAR_OUTPUT
END_VAR
VAR
END_VAR

(*READ HARDWARE FUCNTION BLOCK

	Reads all variables from devices on the EtherCAT network and
	assigns them to their relevant program variables.  This will
	happen every PLC scan*)

(*Left Drive Motor*)
//HARV.DriveSys.DriveLeftIN.ActualVelocity := MOTORS.DriveLeft.ActualVelocity;
HARV.DriveSys.DriveLeftIN.StatusWord 			:= MOTORS.DriveLeft.StatusWord;
HARV.DriveSys.DriveLeftIN.ActualVelocity 		:= MOTORS.DriveLeft.ActualVelocity;
HARV.DriveSys.DriveLeftIN.BatteryVoltage		:= MOTORS.DriveLeft.BatteryVoltage;
HARV.DriveSys.DriveLeftIN.BatteryCurrent		:= MOTORS.DriveLeft.BatteryCurrent;
HARV.DriveSys.DriveLeftIN.HeatSinkTemp			:= MOTORS.DriveLeft.HeatsinkTemp;
HARV.DriveSys.DriveLeftIN.CapacitorVoltage		:= MOTORS.DriveLeft.CapacitorVoltage;

(*Right Drive Motor*)
HARV.DriveSys.DriveRightIN.StatusWord			:= MOTORS.DriveRight.StatusWord;
HARV.DriveSys.DriveRightIN.ActualVelocity 		:= MOTORS.DriveRight.ActualVelocity;
HARV.DriveSys.DriveRightIN.BatteryVoltage		:= MOTORS.DriveRight.BatteryVoltage;
HARV.DriveSys.DriveRightIN.BatteryCurrent		:= MOTORS.DriveRight.BatteryCurrent;
HARV.DriveSys.DriveRightIN.HeatSinkTemp			:= MOTORS.DriveRight.HeatsinkTemp;
HARV.DriveSys.DriveRightIN.CapacitorVoltage		:= MOTORS.DriveRight.CapacitorVoltage;

(*Left Steering Motor*)
HARV.DriveSys.SteerLeftIN.StatusWord 			:= MOTORS.SteerLeft.StatusWord;
HARV.DriveSys.SteerLeftIN.ActualPosition 		:= MOTORS.SteerLeft.ActualPosition;
HARV.DriveSys.SteerLeftIN.ActualVelocity 		:= MOTORS.SteerLeft.ActualVelocity;
HARV.DriveSys.SteerLeftIN.OperationModeDisplay 	:= MOTORS.SteerLeft.OperationModeDisplay;

(*Right Steering Motor*)
HARV.DriveSys.SteerRightIN.StatusWord 			:= MOTORS.SteerRight.StatusWord;
HARV.DriveSys.SteerRightIN.ActualPosition 		:= MOTORS.SteerRight.ActualPosition;
HARV.DriveSys.SteerRightIN.ActualVelocity 		:= MOTORS.SteerRight.ActualVelocity;
HARV.DriveSys.SteerRightIN.OperationModeDisplay := MOTORS.SteerRight.OperationModeDisplay;

(*Left Conveyance Motor*)

(*Right Conveyance Motor*)

(*Tilt Control Inputs*)

(*Digital Inputs EL1018*)
//HARV.DriveSys.JohnButtonInput := IO.DI_SLICE_0[0];
UI.PickButton := IO.DI_SLICE_0[0];
HARV.TiltControl.PressureSwitch := IO.DI_SLICE_0[1];
UI.EStop := IO.DI_SLICE_0[2];

(*Analog Inputs EL3064*)
HARV.DriveSys.JoyStick_X 		:= IO.AI_SLICE_0[0];
HARV.DriveSys.JoyStick_Y 		:= IO.AI_SLICE_0[1];
//HARV.DriveSys.JoyStick_Button 	:= IO.AI_SLICE_0[2];
HARV.TiltControl.IMU_Roll		:= IO.AI_SLICE_0[2];
HARV.TiltControl.IMU_Pitch		:= IO.AI_SLICE_0[3];

(**)

END_FUNCTION_BLOCK

// ---- POUs/FB_WRITE_HW.TcPOU
FUNCTION_BLOCK FB_WRITE_HW
VAR_INPUT
END_VAR
VAR_OUTPUT
END_VAR
VAR
END_VAR

(*WRITE HARDWARE FUCNTION BLOCK

	Writes all program variables in the PLC to their relevant
	hardware devices on the EtherCAT network.  This will happen
	every PLC scan.*)

(*Left Drive Motor - SEVCON*)
MOTORS.DriveLeft.ControlWord		:= HARV.DriveSys.DriveLeft.SEVCON_OUT.ControlWord;
MOTORS.DriveLeft.TargetVelocity		:= HARV.DriveSys.DriveLeft.SEVCON_OUT.TargetVelocity;
MOTORS.DriveLeft.BrakeOutput		:= HARV.DriveSys.DriveLeft.SEVCON_OUT.BrakeOutput;
MOTORS.DriveLeft.ContactorOutput	:= HARV.DriveSys.DriveLeft.SEVCON_OUT.ContactorOutput;

(*Right Drive Motor - SEVCON*)
MOTORS.DriveRight.ControlWord		:= HARV.DriveSys.DriveRight.SEVCON_OUT.ControlWord;
MOTORS.DriveRight.TargetVelocity	:= HARV.DriveSys.DriveRight.SEVCON_OUT.TargetVelocity;
MOTORS.DriveRight.BrakeOutput		:= HARV.DriveSys.DriveRight.SEVCON_OUT.BrakeOutput;
MOTORS.DriveRight.BrakeOutput		:= HARV.DriveSys.DriveRight.SEVCON_OUT.ContactorOutput;

(*Left Steering Motor - PD6*)
MOTORS.SteerLeft.ControlWord		:= HARV.DriveSys.SteerLeft.PD4_OUT.ControlWord;
MOTORS.SteerLeft.OperationMode		:= HARV.DriveSys.SteerLeft.PD4_OUT.OperationMode;
MOTORS.SteerLeft.SubmodeSelect		:= HARV.DriveSys.SteerLeft.PD4_OUT.SubmodeSelect;
MOTORS.SteerLeft.HomingMethod		:= HARV.DriveSys.SteerLeft.PD4_OUT.HomingMethod;
MOTORS.SteerLeft.Polarity			:= HARV.DriveSys.SteerLeft.PD4_OUT.Polarity;
MOTORS.SteerLeft.TargetVelocity		:= HARV.DriveSys.SteerLeft.PD4_OUT.TargetVelocity;
MOTORS.SteerLeft.ProfileVelocity	:= HARV.DriveSys.SteerLeft.PD4_OUT.ProfileVelocity;
MOTORS.SteerLeft.TargetPosition		:= HARV.DriveSys.SteerLeft.PD4_OUT.TargetPosition;
MOTORS.SteerLeft.Accel				:= HARV.DriveSys.SteerLeft.PD4_OUT.Accel;
MOTORS.SteerLeft.Decel				:= HARV.DriveSys.SteerLeft.PD4_OUT.Decel;

(*Right Steering Motor - PD6*)
MOTORS.SteerRight.ControlWord		:= HARV.DriveSys.SteerRight.PD4_OUT.ControlWord;
MOTORS.SteerRight.OperationMode		:= HARV.DriveSys.SteerRight.PD4_OUT.OperationMode;
MOTORS.SteerRight.SubmodeSelect		:= HARV.DriveSys.SteerRight.PD4_OUT.SubmodeSelect;
MOTORS.SteerRight.HomingMethod		:= HARV.DriveSys.SteerRight.PD4_OUT.HomingMethod;
MOTORS.SteerRight.Polarity			:= HARV.DriveSys.SteerRight.PD4_OUT.Polarity;
MOTORS.SteerRight.TargetVelocity	:= HARV.DriveSys.SteerRight.PD4_OUT.TargetVelocity;
MOTORS.SteerRight.ProfileVelocity	:= HARV.DriveSys.SteerRight.PD4_OUT.ProfileVelocity;
MOTORS.SteerRight.TargetPosition	:= HARV.DriveSys.SteerRight.PD4_OUT.TargetPosition;
MOTORS.SteerRight.Accel				:= HARV.DriveSys.SteerRight.PD4_OUT.Accel;
MOTORS.SteerRight.Decel				:= HARV.DriveSys.SteerRight.PD4_OUT.Decel;

(*Left Conveyance Motor*)

(*Right Conveyance Motor*)

(*Digital Outputs EL2008*)
IO.DO_SLICE_0[0] := HARV.TiltControl.RollValveLeft.SolenoidExtend;
IO.DO_SLICE_0[1] := HARV.TiltControl.RollValveLeft.SolenoidRetract;
IO.DO_SLICE_0[2] := HARV.TiltControl.RollValveRight.SolenoidExtend;
IO.DO_SLICE_0[3] := HARV.TiltControl.RollValveRight.SolenoidRetract;
IO.DO_SLICE_0[4] := HARV.TiltControl.PitchValve.SolenoidExtend;
IO.DO_SLICE_0[5] := HARV.TiltControl.PitchValve.SolenoidRetract;
IO.DO_SLICE_0[6] := HARV.TiltControl.PumpContactor;

END_FUNCTION_BLOCK

// ---- POUs/UI Level Function Blocks/FB_FRAMESELECTOR.TcPOU
FUNCTION_BLOCK FB_FRAMESELECTOR
VAR
	//SelectedFrame	: FrameSelect;
	SelectedFrame : INT := 0;
	ShowFrame		: BOOL;
END_VAR

END_FUNCTION_BLOCK

// ---- Test/FB_TILT_TEST.TcPOU
FUNCTION_BLOCK FB_TILT_TEST
VAR_INPUT
END_VAR
VAR_OUTPUT
END_VAR
VAR
END_VAR

END_FUNCTION_BLOCK

// ---- GlobalTextList.TcGTLO
TEXTLIST GlobalTextList
  759 = ''
  183 = '%.0f'
  278 = '%.1f'
  808 = '%2.2f'
  490 = '%3.2f'
  964 = '%4.2f'
  954 = '%s'
  65 = '%S'
  73 = "%s '%'"
  561 = '%s%'
  480 = "%t[ddd MMM dd',' yyyy hh:mm tt]"
  560 = "%t[ddd MMM dd',' yyyy hh:mm:ss tt]"
  888 = '+'
  17 = '+/- TRIM'
  604 = '+5'
  792 = '-'
  397 = '-1.2'
  393 = '40'
  782 = '50%'
  199 = '8.5'
  116 = '<'
  886 = '>'
  203 = 'Acres / Hour'
  48 = 'Apples / Hour'
  826 = 'Auto'
  563 = 'Auto-Level'
  929 = 'Bin Filler'
  143 = 'Bin Filler Adjustments'
  595 = 'Binfiller'
  700 = 'Binfiller Status'
  928 = 'Button 1'
  967 = 'Button 2'
  885 = 'Button 3'
  296 = 'Button 4'
  530 = 'Camera lens dirty'
  887 = 'Color Threshold'
  35 = 'Culling Threshold'
  800 = 'Degrees'
  897 = 'Disable'
  467 = 'Drive Speed'
  256 = 'Drive Speed (Acres / Hr)'
  845 = 'Drive Velocity'
  657 = 'Drive Velocity (m/s)'
  834 = 'Drive Velocity (mm/s)'
  856 = 'Drive: Auto'
  591 = 'Estimated APH'
  171 = 'Front'
  361 = 'IMU Roll Input'
  562 = 'Joystick Position X'
  301 = 'Joystick Position Y'
  181 = 'Left Displacement (in)'
  53 = 'Left Displacement (mm)'
  589 = 'Left Wheel Angle'
  838 = 'Left Wheel Velocity'
  209 = 'Left Wheel Velocity (m/s)'
  466 = 'Left Wheel Velocity (mm/s)'
  395 = 'Low grip success % detected'
  211 = 'Low grip success detected'
  488 = 'Low grip success, check vac'
  128 = 'Lower'
  699 = 'Manual'
  679 = 'Max Bin Fill Height'
  334 = 'Pick Rate'
  762 = 'Pick Rate (Apples / Hr)'
  987 = 'Pitch'
  241 = 'Pitch (+)'
  275 = 'Pitch (-)'
  314 = 'Pitch Angle'
  86 = 'Pump'
  520 = 'Radius of Curvature'
  849 = 'Radius of Curvature (in)'
  955 = 'Raise'
  524 = 'Right Displacement (in)'
  764 = 'Right Displacement (mm)'
  942 = 'Right Wheel Angle'
  758 = 'Right Wheel Velocity'
  889 = 'Right Wheel Velocity (m/s)'
  895 = 'Right Wheel Velocity (mm/s)'
  34 = 'Robot'
  172 = 'Robot 1'
  316 = 'Robot 10'
  930 = 'Robot 11'
  366 = 'Robot 12'
  713 = 'Robot 2'
  313 = 'Robot 3'
  732 = 'Robot 4'
  224 = 'Robot 5'
  39 = 'Robot 6'
  390 = 'Robot 7'
  656 = 'Robot 8'
  593 = 'Robot 89'
  148 = 'Robot 9'
  760 = 'Robot Status'
  547 = 'Roll (+)'
  194 = 'Roll (-)'
  152 = 'Roll Angle'
  450 = 'Slope Angle (Degrees)'
  614 = 'Steering Angle'
  877 = 'W'
  981 = 'Zone 1'
  544 = 'Zone 2'
  277 = 'Zone 3'
  495 = 'Zone 4'
  774 = '^'
END_TEXTLIST

// ---- VISUs/DriveSysTest.TcVIS
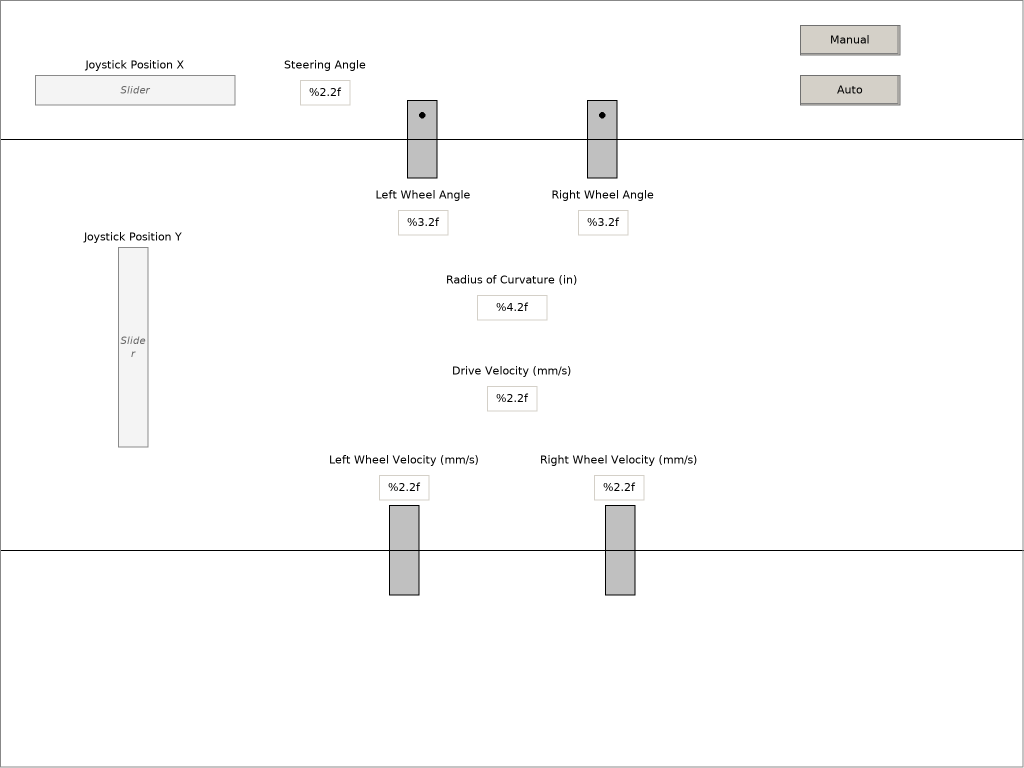
VISUALIZATION DriveSysTest  // 1024x768
    Rectangle (407,100 30x78)
        p2858320360: HARV.DriveSys.LeftWheelAngleCommand
    Rectangle (587,100 30x78)
        p2858320360: HARV.DriveSys.RightWheelAngleCommand
    Rectangle (605,505 30x90)
    Rectangle (389,505 30x90)
    Textfield (398,210 50x25), "%3.2f", text variable: HARV.DriveSys.LeftWheelAngleCommand
    Textfield (578,210 50x25), "%3.2f", text variable: HARV.DriveSys.RightWheelAngleCommand
    Textfield (379,475 50x25), "%2.2f", text variable: HARV.DriveSys.LeftVelCommand
    Textfield (594,475 50x25), "%2.2f", text variable: HARV.DriveSys.RightVelCommand
    Label (348,180 150x30), "Left Wheel Angle"
    Label (528,180 150x30), "Right Wheel Angle"
    Textfield (300,80 50x25), "%2.2f", text variable: HARV.DriveSys.SteeringAngleInput
        OnMouseClick: write the text variable via Default, min -90.0, max 90.0
    Label (250,50 150x30), "Steering Angle"
    Textfield (477,295 70x25), "%4.2f", text variable: HARV.DriveSys.ICC_R
    Label (437,265 150x30), "Radius of Curvature (in)"
    Label (324,445 160x30), "Left Wheel Velocity (mm/s)"
    Label (539,445 160x30), "Right Wheel Velocity (mm/s)"
    Textfield (487,386 50x25), "%2.2f", text variable: HARV.DriveSys.DriveVelInput
        OnMouseClick: write the text variable via Default, min -1.0, max 1.0
    Label (437,356 150x30), "Drive Velocity (mm/s)"
    Slider (35,75 200x30), variable: HARV.DriveSys.JoyStick_X, scale 0..16300
    Label (60,50 150x30), "Joystick Position X"
    Slider (118,247 30x200), variable: HARV.DriveSys.JoyStick_Y, scale 0..16300
    Label (58,222 150x30), "Joystick Position Y"
    Line (-200,139) (1224,139)
        p2858320360: HARV.DriveSys.RightWheelAngleCommand
    Line (-200,139) (1224,139)
        p2858320360: HARV.DriveSys.LeftWheelAngleCommand
    Line (0,550) (1024,550)
    Line (512,550) (512,550)
        p874137650: (HARV.DriveSys.ICC_R)*3
    Ellipse (419,112 6x6)
    Ellipse (599,112 6x6)
    Button (800,25 100x30), "Manual"
        OnMouseClick: toggle HARV.DriveSys.ManualDriveEnable
    Button (800,75 100x30), "Auto"
        OnMouseClick: toggle HARV.DriveSys.AutoDriveEnable
END_VISUALIZATION

// ---- VISUs/Harv UI Components/Home Screen Components/ChassisControls.TcVIS
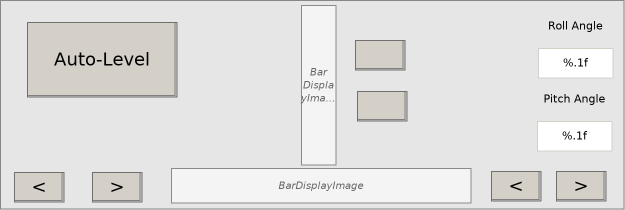
VISUALIZATION ChassisControls  // 625x210
    BarDisplayImage (171,168 300x35), style: BarDisplayImage-Gray, scale format: %.0f, scale -10..10
    BarDisplayImage (301,5 35x160), style: BarDisplayImage-Gray, scale format: %.0f, scale -10..10
    Button (27,22 150x75), "Auto-Level"
    Textfield (538,48 75x30), "%.1f"
    Textfield (537,84 75x30), "Pitch Angle"
    Textfield (538,11 75x30), "Roll Angle"
    Textfield (537,121 75x30), "%.1f"
    Button (14,172 50x30), "<"
    Button (92,172 50x30), ">"
    Button (491,171 50x30), "<"
    Button (556,171 50x30), ">"
    Button (355,40 50x30)
    Button (357,91 50x30)
        p2277200375: -90
END_VISUALIZATION

// ---- VISUs/Harv UI Components/Home Screen Components/DriveControls.TcVIS
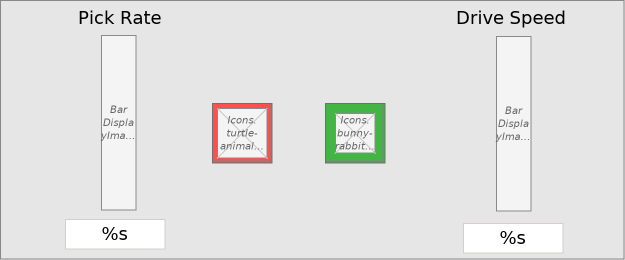
VISUALIZATION DriveControls  // 625x260
    Group (325,103 75x75)
        OnMouseClick: execute { HARV.DriveSys.AutoDriveSpeedCommand := HARV.DriveSys.AutoDriveSpeedCommand + 5; }
        Button (0,0 60x60)
        Image (10,10 40x40), image: Icons.bunny-rabbit-icon
    Group (212,103 75x75)
        OnMouseClick: execute { HARV.DriveSys.AutoDriveSpeedCommand := HARV.DriveSys.AutoDriveSpeedCommand - 5; }
        Button (0,0 60x60)
        Image (5,5 50x50), image: Icons.turtle-animal-icon
    Textfield (65,219 100x30), "%s"
    BarDisplayImage (101,35 35x175), style: BarDisplayImage-Gray, scale format: %.0f, scale 0..100
    BarDisplayImage (496,36 35x175), value: HARV.DriveSys.AutoDriveSpeedActual, style: BarDisplayImage-Gray, scale format: %.1f, scale 0..100
    Textfield (463,223 100x30), "%s", text variable: HARV.DriveSys.AutoDriveSpeedActual
    Textfield (436,3 150x30), "Drive Speed"
    Textfield (45,3 150x30), "Pick Rate"
END_VISUALIZATION

// ---- VISUs/Harv UI Components/Home Screen Components/LeftRobotStatus.TcVIS
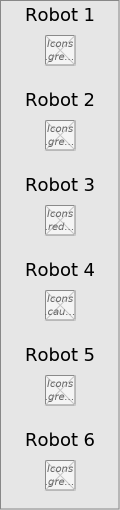
VISUALIZATION LeftRobotStatus  // 120x510
    Textfield (0,0 120x30), "Robot 1"
    Textfield (0,85 120x30), "Robot 2"
    Textfield (0,170 120x30), "Robot 3"
    Textfield (0,255 120x30), "Robot 4"
        OnMouseClick: execute { UI.FrameSelector.SelectedFrame := 1; }
    Textfield (0,340 120x30), "Robot 5"
    Textfield (0,425 120x30), "Robot 6"
    Image (45,35 30x30), input disabled if: TRUE, image: Icons.green-checkmark-icon
    Image (45,120 30x30), image: Icons.green-checkmark-icon
    Image (45,205 30x30), image: Icons.red-x-icon
    Image (45,290 30x30), image: Icons.caution-icon
        OnMouseClick: execute { UI.FrameSelector.SelectedFrame := 1; }
    Image (45,375 30x30), image: Icons.green-checkmark-icon
    Image (45,460 30x30), image: Icons.green-checkmark-icon
END_VISUALIZATION

// ---- VISUs/Harv UI Components/Home Screen Components/RightRobotStatus.TcVIS
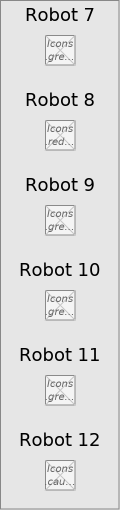
VISUALIZATION RightRobotStatus  // 120x510
    Textfield (0,0 120x30), "Robot 7"
    Textfield (0,85 120x30), "Robot 8"
    Textfield (0,170 120x30), "Robot 9"
    Textfield (0,255 120x30), "Robot 10"
    Textfield (0,340 120x30), "Robot 11"
    Textfield (0,425 120x30), "Robot 12"
    Image (45,35 30x30), input disabled if: TRUE, image: Icons.green-checkmark-icon
    Image (45,120 30x30), colour toggle: TRUE, input disabled if: TRUE, image: Icons.red-x-icon
    Image (45,205 30x30), input disabled if: TRUE, image: Icons.green-checkmark-icon
    Image (45,290 30x30), input disabled if: TRUE, image: Icons.green-checkmark-icon
    Image (45,375 30x30), input disabled if: TRUE, image: Icons.green-checkmark-icon
    Image (45,460 30x30), input disabled if: TRUE, image: Icons.caution-icon
        OnMouseClick: OpenDialog Dialog=VisuDialogs.MessageBox, Parameters={eType: , sMessageTxt: 'Warning Message Here', sTitle: 'WARNING'}, OpenModal=True, PositionX=312, PositionY=100
END_VISUALIZATION

// ---- VISUs/Harv UI Components/Home Screen Components/RobotStatusPopup.TcVIS
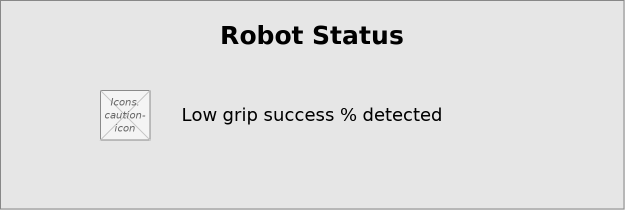
VISUALIZATION RobotStatusPopup  // 625x210
    Textfield (212,10 200x50), "Robot Status"
    Image (100,90 50x50), image: Icons.caution-icon
    Textfield (162,100 300x30), "Low grip success % detected"
END_VISUALIZATION

// ---- VISUs/Harv UI Components/Stats Screen Components/LeftRobotStats.TcVIS
VISUALIZATION LeftRobotStats  // 2x2
END_VISUALIZATION

// ---- VISUs/Harv UI Components/Stats Screen Components/HarvStats.TcVIS
VISUALIZATION HarvStats  // 2x2
END_VISUALIZATION

// ---- VISUs/Harv UI Components/Stats Screen Components/RightRobotStats.TcVIS
VISUALIZATION RightRobotStats  // 2x2
END_VISUALIZATION

// ---- VISUs/Harv UI Components/Supervisor Screen Components/BinFiller.TcVIS
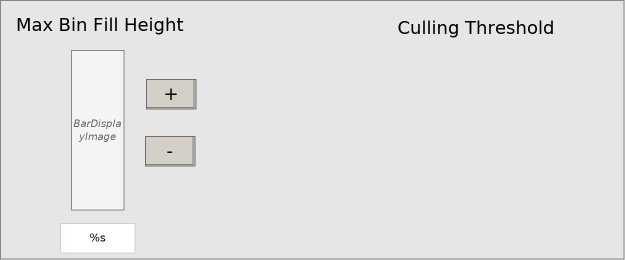
VISUALIZATION BinFiller  // 625x260
    Textfield (0,10 200x30), "Max Bin Fill Height"
    Textfield (60,223 75x30), "%s"
    BarDisplayImage (71,50 53x160), style: BarDisplayImage-Gray, scale format: %.0f, scale 0..100
    Button (146,79 50x30), "+"
    Button (145,136 50x30), "-"
    Textfield (376,13 200x30), "Culling Threshold"
END_VISUALIZATION

// ---- VISUs/Harv UI Components/Supervisor Screen Components/ColorThreshold.TcVIS
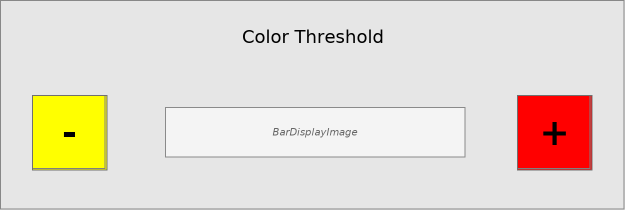
VISUALIZATION ColorThreshold  // 625x210
    Button (517,95 75x75), "+"
    Button (32,95 75x75), "-"
    Textfield (238,22 150x30), "Color Threshold"
    BarDisplayImage (165,107 300x50), style: BarDisplayImage-Gray, scale format: %.1f, scale 0..100
END_VISUALIZATION

// ---- VISUs/Harv UI Components/Supervisor Screen Components/Conveyance.TcVIS
VISUALIZATION Conveyance  // 2x2
END_VISUALIZATION

// ---- VISUs/Harv UI Components/Supervisor Screen Components/LeftRobotControls.TcVIS
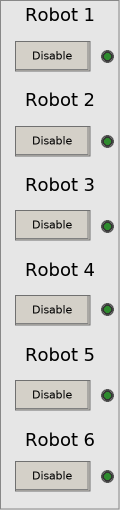
VISUALIZATION LeftRobotControls  // 120x510
    Textfield (0,0 120x30), "Robot 1"
    Textfield (0,85 120x30), "Robot 2"
    Textfield (0,170 120x30), "Robot 3"
    Textfield (0,255 120x30), "Robot 4"
        OnMouseClick: OpenDialog Dialog=VisuDialogs.MessageBox, Parameters={eType: , sMessageTxt: 'Warning Message Here', sTitle: 'WARNING'}, OpenModal=True, PositionX=312, PositionY=100
    Textfield (0,340 120x30), "Robot 5"
    Textfield (0,425 120x30), "Robot 6"
    Button (15,41 75x30), "Disable"
    Button (15,126 75x30), "Disable"
    Button (15,210 75x30), "Disable"
    Button (15,295 75x30), "Disable"
    Button (15,380 75x30), "Disable"
    Button (15,461 75x30), "Disable"
    Lamp1 (100,49 15x15), variable: TRUE, style: Lamp-Lamp1-Green
    Lamp1 (100,134 15x15), variable: TRUE, style: Lamp-Lamp1-Green
    Lamp1 (100,219 15x15), variable: TRUE, style: Lamp-Lamp1-Green
    Lamp1 (100,302 15x15), variable: TRUE, style: Lamp-Lamp1-Green
    Lamp1 (100,388 15x15), variable: TRUE, style: Lamp-Lamp1-Green
    Lamp1 (100,469 15x15), variable: TRUE, style: Lamp-Lamp1-Green
END_VISUALIZATION

// ---- VISUs/Harv UI Components/Supervisor Screen Components/RightRobotControls.TcVIS
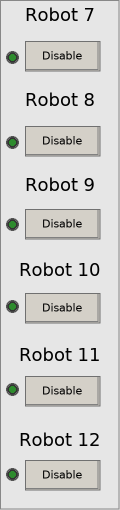
VISUALIZATION RightRobotControls  // 120x510
    Textfield (0,0 120x30), "Robot 7"
    Textfield (0,85 120x30), "Robot 8"
    Textfield (0,170 120x30), "Robot 9"
    Textfield (0,255 120x30), "Robot 10"
    Textfield (0,340 120x30), "Robot 11"
    Textfield (0,425 120x30), "Robot 12"
    Button (25,41 75x30), "Disable"
    Button (25,126 75x30), "Disable"
    Button (25,209 75x30), "Disable"
    Button (25,293 75x30), "Disable"
    Button (25,376 75x30), "Disable"
    Button (25,460 75x30), "Disable"
    Lamp1 (5,50 15x15), variable: TRUE, style: Lamp-Lamp1-Green
    Lamp1 (5,135 15x15), variable: TRUE, style: Lamp-Lamp1-Green
    Lamp1 (5,217 15x15), variable: TRUE, style: Lamp-Lamp1-Green
    Lamp1 (5,299 15x15), variable: TRUE, style: Lamp-Lamp1-Green
    Lamp1 (5,382 15x15), variable: TRUE, style: Lamp-Lamp1-Green
    Lamp1 (5,467 15x15), variable: TRUE, style: Lamp-Lamp1-Green
END_VISUALIZATION

// ---- VISUs/Harv UI Components/Home_Screen.TcVIS
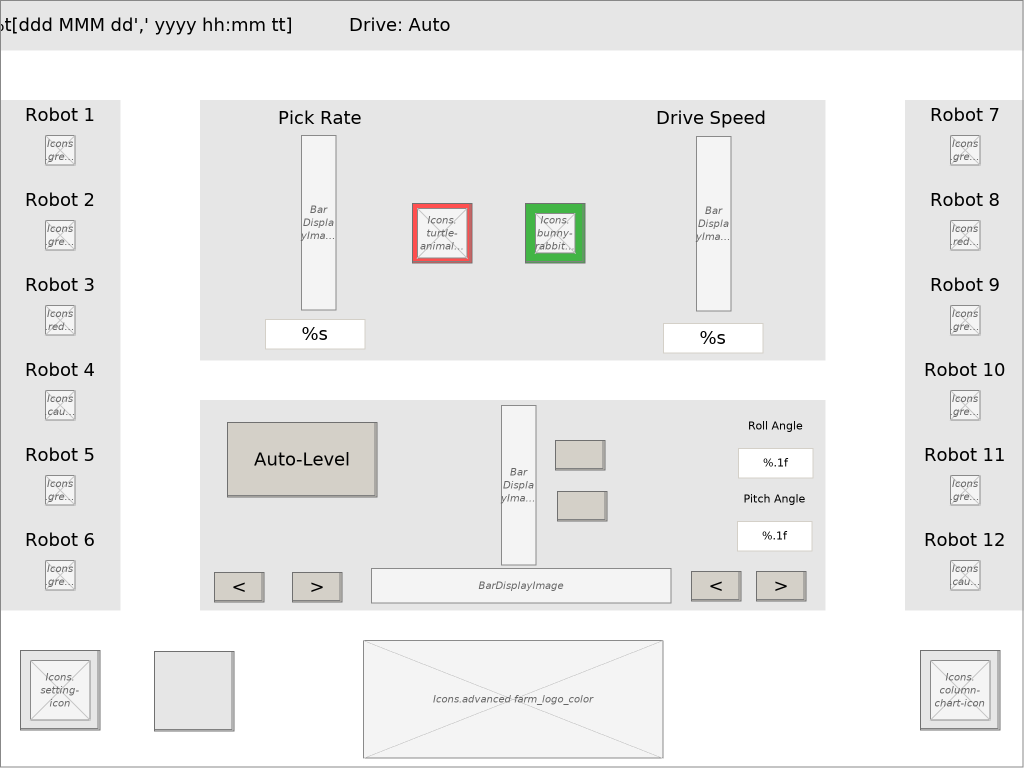
VISUALIZATION Home_Screen  // 1024x768
    Rectangle (905,100 120x510)
    Rectangle (0,100 120x510)
    Rectangle (200,400 625x210)
    Rectangle (200,100 625x260)
    Rectangle (0,0 1024x50)
    Frame (0,0 1024x50)
        shows StatusBar()
    Image (363,640 300x118), image: Icons.advanced farm_logo_color
    Group (20,650 80x80)
        OnMouseClick: change screen: Supervisor_Screen
        Button (0,0 80x80)
        Image (10,10 60x60), image: Icons.setting-icon
    Group (920,650 80x80)
        OnMouseClick: change screen: Stats_Screen
        Button (0,0 80x80)
        Image (10,10 60x60), image: Icons.column-chart-icon
    Frame (200,400 625x210), frame switch variable: UI.FrameSelector.SelectedFrame
        shows ChassisControls()
        shows RobotStatusPopup()
    Frame (200,100 625x260)
        shows DriveControls()
    Frame (0,100 120x510)
        shows LeftRobotStatus()
    Frame (905,100 120x510)
        shows RightRobotStatus()
    Button (154,651 80x80)
END_VISUALIZATION

// ---- VISUs/Harv UI Components/Stats_Screen.TcVIS
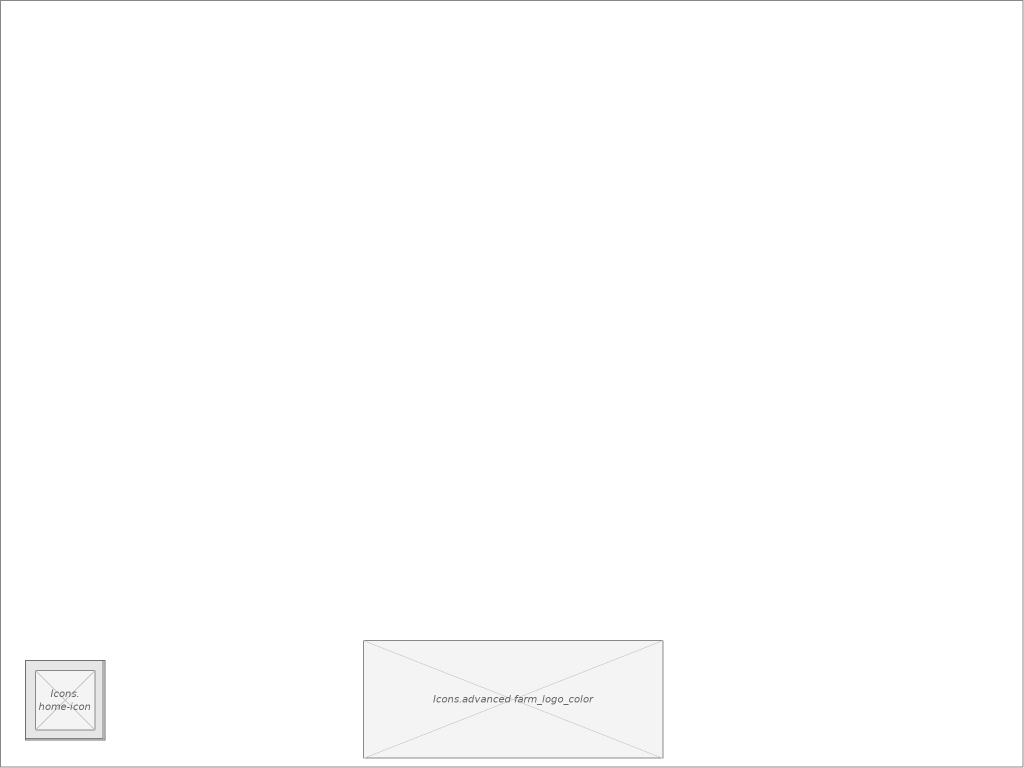
VISUALIZATION Stats_Screen  // 1024x768
    Image (363,640 300x118), image: Icons.advanced farm_logo_color
    Group (25,660 80x80)
        OnMouseClick: change screen: Home_Screen
        Button (0,0 80x80)
        Image (10,10 60x60), image: Icons.home-icon
END_VISUALIZATION

// ---- VISUs/Harv UI Components/StatusBar.TcVIS
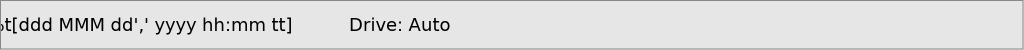
VISUALIZATION StatusBar  // 1024x50
    Textfield (-35,0 350x50), "%t[ddd MMM dd',' yyyy hh:mm tt]", text variable: HARV.TimeTracker.TimeStampStruct
    Textfield (325,0 150x50), "Drive: Auto"
END_VISUALIZATION

// ---- VISUs/Harv UI Components/Supervisor_Screen.TcVIS
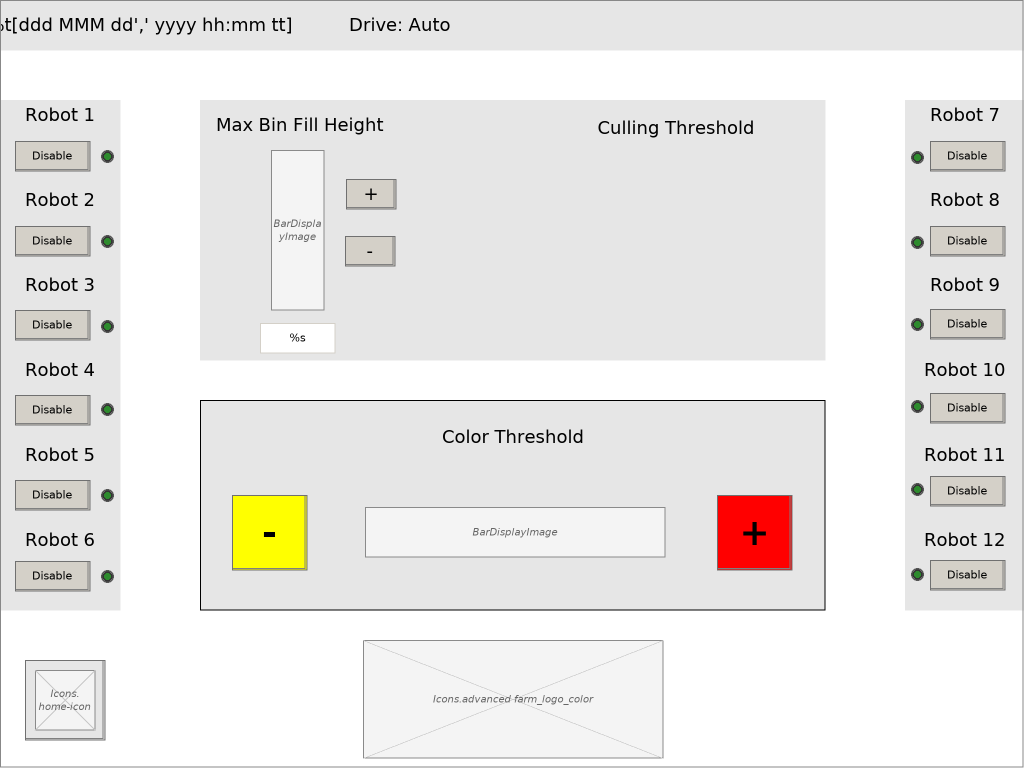
VISUALIZATION Supervisor_Screen  // 1024x768
    Frame (0,0 1024x50)
        shows StatusBar()
    Group (25,660 80x80)
        OnMouseClick: change screen: Home_Screen
        Button (0,0 80x80)
        Image (10,10 60x60), image: Icons.home-icon
    Image (363,640 300x118), image: Icons.advanced farm_logo_color
    Rectangle (200,100 625x260)
    Rectangle (905,100 120x510)
    Rectangle (0,100 120x510)
    Frame (0,100 120x510)
        shows LeftRobotControls()
    Frame (905,100 120x510)
        shows RightRobotControls()
    Frame (200,400 625x210)
        shows ColorThreshold()
    Frame (200,100 625x260)
        shows BinFiller()
    Rectangle (200,400 625x210)
END_VISUALIZATION

// ---- VISUs/TiltControlTest.TcVIS
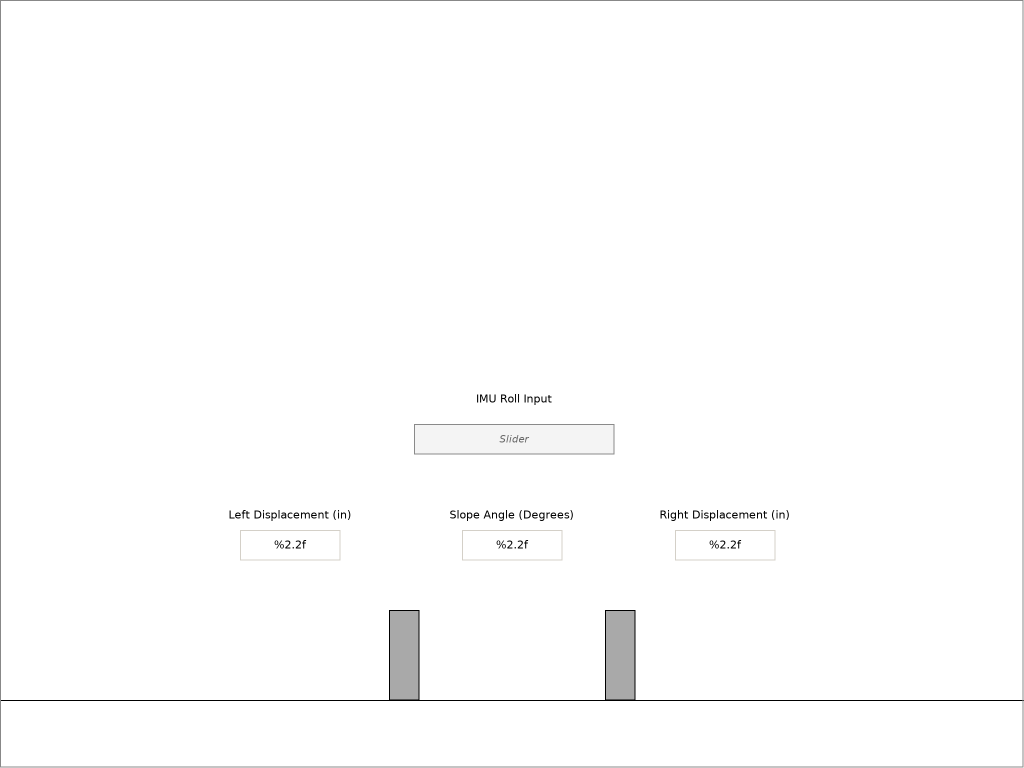
VISUALIZATION TiltControlTest  // 1024x768
    Line (0,700) (1024,700)
        p2858320360: HARV.TiltControl.SlopeAngle
        p2738717112: (HARV.TiltControl.TiltDisplacement * 3) / 2
    Rectangle (389,610 30x90)
        p2738717112: HARV.TiltControl.TiltLeftDisplacement *3
    Rectangle (605,610 30x90)
        p2738717112: HARV.TiltControl.TiltRightDisplacement * 3
    Group (437,500 150x60)
        Textfield (25,30 100x30), "%2.2f", text variable: HARV.TiltControl.SlopeAngle
            OnMouseClick: write the text variable via Default, min -10, max 10
        Label (0,0 150x30), "Slope Angle (Degrees)"
    Group (650,500 150x60)
        Textfield (25,30 100x30), "%2.2f", text variable: HARV.TiltControl.TiltRightDisplacement
            OnMouseClick: write the text variable via Default, min -10, max 10
        Label (0,0 150x30), "Right Displacement (in)"
    Group (215,500 150x60)
        Textfield (25,30 100x30), "%2.2f", text variable: HARV.TiltControl.TiltLeftDisplacement
            OnMouseClick: write the text variable via Default, min -10, max 10
        Label (0,0 150x30), "Left Displacement (in)"
    Slider (414,424 200x30), variable: HARV.TiltControl.IMU_Roll, scale -11..11
    Label (439,384 150x30), "IMU Roll Input"
END_VISUALIZATION
